LIN {X 0,Y 285.756,Z 658.565,A -85,B 0,C 180,E1 17474.349,E2 17474.349} C_VEL
LIN {X 0,Y 305.799,Z 701.656,A -85,B 0,C 180,E1 17484.152,E2 17484.152} C_VEL
LIN {X 0,Y 312.172,Z 727.073,A -85,B 0,C 180,E1 17488.423,E2 17488.423} C_VEL
LIN {X 0,Y 292.235,Z 787.027,A -85,B 0,C 180,E1 17493.812,E2 17493.812} C_VEL
LIN {X 0,Y 268.974,Z 838.866,A -85,B 0,C 180,E1 17502.314,E2 17502.314} C_VEL
LIN {X 0,Y 248.662,Z 880.297,A -85,B 0,C 180,E1 17514.564,E2 17514.564} C_VEL
LIN {X 0,Y 238.211,Z 907.781,A -85,B 0,C 180,E1 17529.488,E2 17529.488} C_VEL
LIN {X 0,Y 236.533,Z 919.61,A -85,B 0,C 180,E1 17543.125,E2 17543.125} C_VEL
LIN {X 0,Y 236.659,Z 920.093,A -85,B 0,C 180,E1 17555.518,E2 17555.518} C_VEL
LIN {X 0,Y 237.841,Z 908.97,A -85,B 0,C 180,E1 17569.569,E2 17569.569} C_VEL
LIN {X 0,Y 247.611,Z 883.003,A -85,B 0,C 180,E1 17584.7,E2 17584.7} C_VEL
LIN {X 0,Y 269.348,Z 841.838,A -85,B 0,C 180,E1 17597.744,E2 17597.744} C_VEL
LIN {X 0,Y 295.092,Z 790.298,A -85,B 0,C 180,E1 17606.682,E2 17606.682} C_VEL
LIN {X 0,Y 317.64,Z 730.915,A -85,B 0,C 180,E1 17612.277,E2 17612.277} C_VEL
LIN {X 0,Y 319.176,Z 721.636,A -85,B 0,C 180,E1 17613.218,E2 17613.218} C_VEL
LIN {X 0,Y 311.516,Z 690.262,A -85,B 0,C 180,E1 17620.895,E2 17620.895} C_VEL
LIN {X 0,Y 304.486,Z 672.096,A -85,B 0,C 180,E1 17629.77,E2 17629.77} C_VEL
LIN {X 0,Y 300.924,Z 676.866,A -85,B 0,C 180,E1 17636.437,E2 17636.437} C_VEL
LIN {X 0,Y 302.486,Z 683.644,A -85,B 0,C 180,E1 17643.411,E2 17643.411} C_VEL
LIN {X 0,Y 306.536,Z 706.136,A -85,B 0,C 180,E1 17652.005,E2 17652.005} C_VEL
LIN {X 0,Y 306.21,Z 719.511,A -85,B 0,C 180,E1 17654.903,E2 17654.903} C_VEL
LIN {X 0,Y 283.493,Z 770.529,A -85,B 0,C 180,E1 17660.967,E2 17660.967} C_VEL
LIN {X 0,Y 260.071,Z 809.733,A -85,B 0,C 180,E1 17669.993,E2 17669.993} C_VEL
LIN {X 0,Y 241.204,Z 836.353,A -85,B 0,C 180,E1 17682.29,E2 17682.29} C_VEL
LIN {X 0,Y 231.777,Z 848.177,A -85,B 0,C 180,E1 17696.186,E2 17696.186} C_VEL
LIN {X 0,Y 230.704,Z 847.604,A -85,B 0,C 180,E1 17708.792,E2 17708.792} C_VEL
LIN {X 0,Y 237.274,Z 834.196,A -85,B 0,C 180,E1 17722.816,E2 17722.816} C_VEL
LIN {X 0,Y 252.204,Z 806.032,A -85,B 0,C 180,E1 17735.424,E2 17735.424} C_VEL
LIN {X 0,Y 272.012,Z 764.995,A -85,B 0,C 180,E1 17744.744,E2 17744.744} C_VEL
LIN {X 0,Y 290.785,Z 713.245,A -85,B 0,C 180,E1 17751.027,E2 17751.027} C_VEL
LIN {X 0,Y 292.766,Z 701.675,A -85,B 0,C 180,E1 17752.282,E2 17752.282} C_VEL
LIN {X 0,Y 279.473,Z 664.949,A -85,B 0,C 180,E1 17761.189,E2 17761.189} C_VEL
LIN {X 0,Y 262.364,Z 636.414,A -85,B 0,C 180,E1 17772.063,E2 17772.063} C_VEL
LIN {X 0,Y 249.885,Z 618.017,A -85,B 0,C 180,E1 17784.7,E2 17784.7} C_VEL
LIN {X 0,Y 246.642,Z 613.282,A -85,B 0,C 180,E1 17801.641,E2 17801.641} C_VEL
LIN {X 0,Y 253.782,Z 621.283,A -85,B 0,C 180,E1 17813.984,E2 17813.984} C_VEL
LIN {X 0,Y 263.474,Z 634.294,A -85,B 0,C 180,E1 17822.404,E2 17822.404} C_VEL
LIN {X 0,Y 282.574,Z 665.228,A -85,B 0,C 180,E1 17833.721,E2 17833.721} C_VEL
LIN {X 0,Y 300.675,Z 706.247,A -85,B 0,C 180,E1 17843.349,E2 17843.349} C_VEL
LIN {X 0,Y 306.304,Z 729.368,A -85,B 0,C 180,E1 17847.452,E2 17847.452} C_VEL
LIN {X 0,Y 285.771,Z 788.355,A -85,B 0,C 180,E1 17852.891,E2 17852.891} C_VEL
LIN {X 0,Y 262.152,Z 838.88,A -85,B 0,C 180,E1 17861.401,E2 17861.401} C_VEL
LIN {X 0,Y 240.939,Z 880.256,A -85,B 0,C 180,E1 17874.076,E2 17874.076} C_VEL
LIN {X 0,Y 230.174,Z 907.605,A -85,B 0,C 180,E1 17889.748,E2 17889.748} C_VEL
LIN {X 0,Y 228.679,Z 918.896,A -85,B 0,C 180,E1 17904.286,E2 17904.286} C_VEL
LIN {X 0,Y 228.733,Z 918.872,A -85,B 0,C 180,E1 17915.71,E2 17915.71} C_VEL
LIN {X 0,Y 229.978,Z 907.706,A -85,B 0,C 180,E1 17930.267,E2 17930.267} C_VEL
LIN {X 0,Y 240.807,Z 881.536,A -85,B 0,C 180,E1 17945.935,E2 17945.935} C_VEL
LIN {X 0,Y 263.596,Z 840.67,A -85,B 0,C 180,E1 17959.097,E2 17959.097} C_VEL
LIN {X 0,Y 290.556,Z 789.057,A -85,B 0,C 180,E1 17968.069,E2 17968.069} C_VEL
LIN {X 0,Y 313.57,Z 730.598,A -85,B 0,C 180,E1 17973.545,E2 17973.545} C_VEL
LIN {X 0,Y 311.052,Z 707.647,A -85,B 0,C 180,E1 17978.228,E2 17978.228} C_VEL
LIN {X 0,Y 303.827,Z 684.399,A -85,B 0,C 180,E1 17986.891,E2 17986.891} C_VEL
LIN {X 0,Y 300.918,Z 677.004,A -85,B 0,C 180,E1 17994.813,E2 17994.813} C_VEL
LIN {X 0,Y 300.924,Z 676.866,A -85,B 0,C 180,E1 17996.437,E2 17996.437} C_VEL
LIN {X 0,Y 299.494,Z 690.532,A -85,B 0,C 180,E1 18002.762,E2 18002.762} C_VEL
LIN {X 0,Y 302.297,Z 710.977,A -85,B 0,C 180,E1 18011.066,E2 18011.066} C_VEL
LIN {X 0,Y 301.828,Z 722.39,A -85,B 0,C 180,E1 18013.737,E2 18013.737} C_VEL
LIN {X 0,Y 278.895,Z 771.501,A -85,B 0,C 180,E1 18019.625,E2 18019.625} C_VEL
LIN {X 0,Y 254.375,Z 810.659,A -85,B 0,C 180,E1 18028.68,E2 18028.68} C_VEL
LIN {X 0,Y 234.95,Z 836.493,A -85,B 0,C 180,E1 18040.585,E2 18040.585} C_VEL
LIN {X 0,Y 224.337,Z 849.161,A -85,B 0,C 180,E1 18054.904,E2 18054.904} C_VEL
LIN {X 0,Y 223.072,Z 848.185,A -85,B 0,C 180,E1 18070.116,E2 18070.116} C_VEL
LIN {X 0,Y 230.402,Z 834.015,A -85,B 0,C 180,E1 18084.332,E2 18084.332} C_VEL
LIN {X 0,Y 246.032,Z 806.043,A -85,B 0,C 180,E1 18096.737,E2 18096.737} C_VEL
LIN {X 0,Y 266.699,Z 764.716,A -85,B 0,C 180,E1 18106.106,E2 18106.106} C_VEL
LIN {X 0,Y 286.019,Z 712.916,A -85,B 0,C 180,E1 18112.334,E2 18112.334} C_VEL
LIN {X 0,Y 286.388,Z 701.757,A -85,B 0,C 180,E1 18114.013,E2 18114.013} C_VEL
LIN {X 0,Y 273.45,Z 666.448,A -85,B 0,C 180,E1 18123.313,E2 18123.313} C_VEL
LIN {X 0,Y 257.524,Z 639.288,A -85,B 0,C 180,E1 18134.83,E2 18134.83} C_VEL
LIN {X 0,Y 247.315,Z 625.136,A -85,B 0,C 180,E1 18147.059,E2 18147.059} C_VEL
LIN {X 0,Y 245.601,Z 621.305,A -85,B 0,C 180,E1 18161.71,E2 18161.71} C_VEL
LIN {X 0,Y 252.429,Z 629.123,A -85,B 0,C 180,E1 18173.688,E2 18173.688} C_VEL
LIN {X 0,Y 263.127,Z 644.042,A -85,B 0,C 180,E1 18183.035,E2 18183.035} C_VEL
LIN {X 0,Y 281.121,Z 675.674,A -85,B 0,C 180,E1 18194.191,E2 18194.191} C_VEL
LIN {X 0,Y 297.749,Z 717.835,A -85,B 0,C 180,E1 18203.991,E2 18203.991} C_VEL
LIN {X 0,Y 300.028,Z 733.449,A -85,B 0,C 180,E1 18206.564,E2 18206.564} C_VEL
LIN {X 0,Y 277.496,Z 793.955,A -85,B 0,C 180,E1 18212.487,E2 18212.487} C_VEL
LIN {X 0,Y 252.286,Z 844.934,A -85,B 0,C 180,E1 18221.893,E2 18221.893} C_VEL
LIN {X 0,Y 231.41,Z 884.207,A -85,B 0,C 180,E1 18235.349,E2 18235.349} C_VEL
LIN {X 0,Y 221.734,Z 909.528,A -85,B 0,C 180,E1 18252.061,E2 18252.061} C_VEL
LIN {X 0,Y 220.778,Z 917.691,A -85,B 0,C 180,E1 18264.239,E2 18264.239} C_VEL
LIN {X 0,Y 220.79,Z 917.646,A -85,B 0,C 180,E1 18275.916,E2 18275.916} C_VEL
LIN {X 0,Y 222.201,Z 906.459,A -85,B 0,C 180,E1 18291.009,E2 18291.009} C_VEL
LIN {X 0,Y 233.986,Z 880.303,A -85,B 0,C 180,E1 18307.148,E2 18307.148} C_VEL
LIN {X 0,Y 258.018,Z 839.639,A -85,B 0,C 180,E1 18320.481,E2 18320.481} C_VEL
LIN {X 0,Y 285.967,Z 788.348,A -85,B 0,C 180,E1 18329.436,E2 18329.436} C_VEL
LIN {X 0,Y 309.296,Z 729.164,A -85,B 0,C 180,E1 18335.183,E2 18335.183} C_VEL
LIN {X 0,Y 304.166,Z 701.793,A -85,B 0,C 180,E1 18342.646,E2 18342.646} C_VEL
LIN {X 0,Y 299.965,Z 687.774,A -85,B 0,C 180,E1 18349.861,E2 18349.861} C_VEL
LIN {X 0,Y 298.698,Z 685.744,A -85,B 0,C 180,E1 18358.601,E2 18358.601} C_VEL
LIN {X 0,Y 299.494,Z 690.532,A -85,B 0,C 180,E1 18362.762,E2 18362.762} C_VEL
LIN {X 0,Y 297.796,Z 710.81,A -85,B 0,C 180,E1 18368.411,E2 18368.411} C_VEL
LIN {X 0,Y 296.984,Z 726.69,A -85,B 0,C 180,E1 18372.665,E2 18372.665} C_VEL
LIN {X 0,Y 272.134,Z 776.524,A -85,B 0,C 180,E1 18378.912,E2 18378.912} C_VEL
LIN {X 0,Y 246.056,Z 815.395,A -85,B 0,C 180,E1 18388.594,E2 18388.594} C_VEL
LIN {X 0,Y 225.73,Z 840.486,A -85,B 0,C 180,E1 18401.706,E2 18401.706} C_VEL
LIN {X 0,Y 216.947,Z 850.083,A -85,B 0,C 180,E1 18413.651,E2 18413.651} C_VEL
LIN {X 0,Y 214.574,Z 850.715,A -85,B 0,C 180,E1 18427.111,E2 18427.111} C_VEL
LIN {X 0,Y 220.669,Z 839.38,A -85,B 0,C 180,E1 18441.914,E2 18441.914} C_VEL
LIN {X 0,Y 235.858,Z 813.54,A -85,B 0,C 180,E1 18455.54,E2 18455.54} C_VEL
LIN {X 0,Y 256.152,Z 775.907,A -85,B 0,C 180,E1 18465.463,E2 18465.463} C_VEL
LIN {X 0,Y 276.694,Z 726.885,A -85,B 0,C 180,E1 18472.365,E2 18472.365} C_VEL
LIN {X 0,Y 281.668,Z 708.955,A -85,B 0,C 180,E1 18474.219,E2 18474.219} C_VEL
LIN {X 0,Y 270.443,Z 674.474,A -85,B 0,C 180,E1 18483.46,E2 18483.46} C_VEL
LIN {X 0,Y 255.662,Z 646.909,A -85,B 0,C 180,E1 18495.168,E2 18495.168} C_VEL
LIN {X 0,Y 246.004,Z 632.903,A -85,B 0,C 180,E1 18507.493,E2 18507.493} C_VEL
LIN {X 0,Y 244.573,Z 629.3,A -85,B 0,C 180,E1 18521.809,E2 18521.809} C_VEL
LIN {X 0,Y 251.076,Z 636.937,A -85,B 0,C 180,E1 18533.379,E2 18533.379} C_VEL
LIN {X 0,Y 262.218,Z 653.044,A -85,B 0,C 180,E1 18543.357,E2 18543.357} C_VEL
LIN {X 0,Y 279.482,Z 686.4,A -85,B 0,C 180,E1 18554.778,E2 18554.778} C_VEL
LIN {X 0,Y 293.957,Z 728.626,A -85,B 0,C 180,E1 18564.483,E2 18564.483} C_VEL
LIN {X 0,Y 293.002,Z 739.507,A -85,B 0,C 180,E1 18565.829,E2 18565.829} C_VEL
LIN {X 0,Y 270.413,Z 796.506,A -85,B 0,C 180,E1 18571.696,E2 18571.696} C_VEL
LIN {X 0,Y 244.727,Z 846.193,A -85,B 0,C 180,E1 18581.271,E2 18581.271} C_VEL
LIN {X 0,Y 223.718,Z 883.939,A -85,B 0,C 180,E1 18594.788,E2 18594.788} C_VEL
LIN {X 0,Y 213.898,Z 908.137,A -85,B 0,C 180,E1 18611.38,E2 18611.38} C_VEL
LIN {X 0,Y 212.809,Z 916.386,A -85,B 0,C 180,E1 18623.858,E2 18623.858} C_VEL
LIN {X 0,Y 212.842,Z 916.424,A -85,B 0,C 180,E1 18636.137,E2 18636.137} C_VEL
LIN {X 0,Y 214.121,Z 906.378,A -85,B 0,C 180,E1 18650.752,E2 18650.752} C_VEL
LIN {X 0,Y 226.469,Z 880.45,A -85,B 0,C 180,E1 18667.808,E2 18667.808} C_VEL
LIN {X 0,Y 251.768,Z 839.926,A -85,B 0,C 180,E1 18681.619,E2 18681.619} C_VEL
LIN {X 0,Y 281.142,Z 788.507,A -85,B 0,C 180,E1 18690.754,E2 18690.754} C_VEL
LIN {X 0,Y 304.387,Z 732.594,A -85,B 0,C 180,E1 18696.267,E2 18696.267} C_VEL
LIN {X 0,Y 300.184,Z 706.471,A -85,B 0,C 180,E1 18703.921,E2 18703.921} C_VEL
LIN {X 0,Y 296.811,Z 694.336,A -85,B 0,C 180,E1 18711.2,E2 18711.2} C_VEL
LIN {X 0,Y 296.088,Z 693.324,A -85,B 0,C 180,E1 18718.588,E2 18718.588} C_VEL
LIN {X 0,Y 297.437,Z 706.176,A -85,B 0,C 180,E1 18726.645,E2 18726.645} C_VEL
LIN {X 0,Y 297.796,Z 710.81,A -85,B 0,C 180,E1 18728.411,E2 18728.411} C_VEL
LIN {X 0,Y 295.364,Z 723.191,A -85,B 0,C 180,E1 18730.755,E2 18730.755} C_VEL
LIN {X 0,Y 288.736,Z 738.824,A -85,B 0,C 180,E1 18732.316,E2 18732.316} C_VEL
LIN {X 0,Y 262.641,Z 785.694,A -85,B 0,C 180,E1 18738.979,E2 18738.979} C_VEL
LIN {X 0,Y 236.659,Z 821.229,A -85,B 0,C 180,E1 18749.008,E2 18749.008} C_VEL
LIN {X 0,Y 216.724,Z 843.948,A -85,B 0,C 180,E1 18762.677,E2 18762.677} C_VEL
LIN {X 0,Y 207.622,Z 852.599,A -85,B 0,C 180,E1 18777.309,E2 18777.309} C_VEL
LIN {X 0,Y 208.233,Z 848.927,A -85,B 0,C 180,E1 18793.399,E2 18793.399} C_VEL
LIN {X 0,Y 218.395,Z 831.675,A -85,B 0,C 180,E1 18808.674,E2 18808.674} C_VEL
LIN {X 0,Y 237.945,Z 799.409,A -85,B 0,C 180,E1 18821.498,E2 18821.498} C_VEL
LIN {X 0,Y 261.063,Z 754.132,A -85,B 0,C 180,E1 18830.5,E2 18830.5} C_VEL
LIN {X 0,Y 276,Z 711.618,A -85,B 0,C 180,E1 18835.458,E2 18835.458} C_VEL
LIN {X 0,Y 265.972,Z 679.01,A -85,B 0,C 180,E1 18844.683,E2 18844.683} C_VEL
LIN {X 0,Y 252.607,Z 653.366,A -85,B 0,C 180,E1 18856.406,E2 18856.406} C_VEL
LIN {X 0,Y 244.487,Z 640.557,A -85,B 0,C 180,E1 18868.092,E2 18868.092} C_VEL
LIN {X 0,Y 243.496,Z 637.271,A -85,B 0,C 180,E1 18881.78,E2 18881.78} C_VEL
LIN {X 0,Y 249.831,Z 645.112,A -85,B 0,C 180,E1 18893.374,E2 18893.374} C_VEL
LIN {X 0,Y 260.201,Z 661.255,A -85,B 0,C 180,E1 18903.174,E2 18903.174} C_VEL
LIN {X 0,Y 275.808,Z 693.161,A -85,B 0,C 180,E1 18914.267,E2 18914.267} C_VEL
LIN {X 0,Y 289.1,Z 735.715,A -85,B 0,C 180,E1 18924.293,E2 18924.293} C_VEL
LIN {X 0,Y 265.502,Z 794.732,A -85,B 0,C 180,E1 18930.261,E2 18930.261} C_VEL
LIN {X 0,Y 238.86,Z 844.483,A -85,B 0,C 180,E1 18939.809,E2 18939.809} C_VEL
LIN {X 0,Y 216.77,Z 882.281,A -85,B 0,C 180,E1 18953.481,E2 18953.481} C_VEL
LIN {X 0,Y 206.069,Z 906.722,A -85,B 0,C 180,E1 18970.645,E2 18970.645} C_VEL
LIN {X 0,Y 204.869,Z 915.125,A -85,B 0,C 180,E1 18983.619,E2 18983.619} C_VEL
LIN {X 0,Y 204.89,Z 915.198,A -85,B 0,C 180,E1 18996.377,E2 18996.377} C_VEL
LIN {X 0,Y 206.365,Z 905.146,A -85,B 0,C 180,E1 19011.57,E2 19011.57} C_VEL
LIN {X 0,Y 219.047,Z 880.402,A -85,B 0,C 180,E1 19028.57,E2 19028.57} C_VEL
LIN {X 0,Y 245.447,Z 840.432,A -85,B 0,C 180,E1 19042.749,E2 19042.749} C_VEL
LIN {X 0,Y 275.715,Z 790.077,A -85,B 0,C 180,E1 19051.919,E2 19051.919} C_VEL
LIN {X 0,Y 299.55,Z 735.967,A -85,B 0,C 180,E1 19057.414,E2 19057.414} C_VEL
LIN {X 0,Y 296.354,Z 711.703,A -85,B 0,C 180,E1 19065.079,E2 19065.079} C_VEL
LIN {X 0,Y 293.659,Z 700.98,A -85,B 0,C 180,E1 19072.637,E2 19072.637} C_VEL
LIN {X 0,Y 293.308,Z 701.695,A -85,B 0,C 180,E1 19079.686,E2 19079.686} C_VEL
LIN {X 0,Y 293.87,Z 718.198,A -85,B 0,C 180,E1 19088.218,E2 19088.218} C_VEL
LIN {X 0,Y 292.904,Z 729.47,A -85,B 0,C 180,E1 19091.416,E2 19091.416} C_VEL
LIN {X 0,Y 288.736,Z 738.824,A -85,B 0,C 180,E1 19092.316,E2 19092.316} C_VEL
LIN {X 0,Y 270.495,Z 767.731,A -85,B 0,C 180,E1 19094.242,E2 19094.242} C_VEL
LIN {X 0,Y 241.389,Z 809.699,A -85,B 0,C 180,E1 19103.087,E2 19103.087} C_VEL
LIN {X 0,Y 216.003,Z 838.571,A -85,B 0,C 180,E1 19116.109,E2 19116.109} C_VEL
LIN {X 0,Y 201.698,Z 852.529,A -85,B 0,C 180,E1 19132.289,E2 19132.289} C_VEL
LIN {X 0,Y 199.239,Z 852.145,A -85,B 0,C 180,E1 19149.958,E2 19149.958} C_VEL
LIN {X 0,Y 207.662,Z 838.172,A -85,B 0,C 180,E1 19165.996,E2 19165.996} C_VEL
LIN {X 0,Y 225.755,Z 810.237,A -85,B 0,C 180,E1 19179.676,E2 19179.676} C_VEL
LIN {X 0,Y 249.087,Z 769.143,A -85,B 0,C 180,E1 19189.579,E2 19189.579} C_VEL
LIN {X 0,Y 270.747,Z 716.234,A -85,B 0,C 180,E1 19196.272,E2 19196.272} C_VEL
LIN {X 0,Y 261.838,Z 684.683,A -85,B 0,C 180,E1 19205.577,E2 19205.577} C_VEL
LIN {X 0,Y 249.851,Z 660.2,A -85,B 0,C 180,E1 19217.308,E2 19217.308} C_VEL
LIN {X 0,Y 243.013,Z 648.329,A -85,B 0,C 180,E1 19228.416,E2 19228.416} C_VEL
LIN {X 0,Y 242.244,Z 645.163,A -85,B 0,C 180,E1 19241.682,E2 19241.682} C_VEL
LIN {X 0,Y 248.26,Z 652.931,A -85,B 0,C 180,E1 19253.134,E2 19253.134} C_VEL
LIN {X 0,Y 258.601,Z 670.439,A -85,B 0,C 180,E1 19263.509,E2 19263.509} C_VEL
LIN {X 0,Y 273.157,Z 703.222,A -85,B 0,C 180,E1 19274.717,E2 19274.717} C_VEL
LIN {X 0,Y 283.014,Z 739.353,A -85,B 0,C 180,E1 19283.325,E2 19283.325} C_VEL
LIN {X 0,Y 258.862,Z 796.578,A -85,B 0,C 180,E1 19289.293,E2 19289.293} C_VEL
LIN {X 0,Y 231.377,Z 845.745,A -85,B 0,C 180,E1 19299.111,E2 19299.111} C_VEL
LIN {X 0,Y 208.218,Z 883.681,A -85,B 0,C 180,E1 19313.765,E2 19313.765} C_VEL
LIN {X 0,Y 197.836,Z 907.082,A -85,B 0,C 180,E1 19331.838,E2 19331.838} C_VEL
LIN {X 0,Y 196.92,Z 913.86,A -85,B 0,C 180,E1 19343.36,E2 19343.36} C_VEL
LIN {X 0,Y 196.939,Z 913.978,A -85,B 0,C 180,E1 19356.635,E2 19356.635} C_VEL
LIN {X 0,Y 198.618,Z 903.937,A -85,B 0,C 180,E1 19372.439,E2 19372.439} C_VEL
LIN {X 0,Y 213.893,Z 877.227,A -85,B 0,C 180,E1 19391.013,E2 19391.013} C_VEL
LIN {X 0,Y 242.601,Z 836.075,A -85,B 0,C 180,E1 19405.182,E2 19405.182} C_VEL
LIN {X 0,Y 273.786,Z 785.568,A -85,B 0,C 180,E1 19413.936,E2 19413.936} C_VEL
LIN {X 0,Y 294.864,Z 739.603,A -85,B 0,C 180,E1 19418.541,E2 19418.541} C_VEL
LIN {X 0,Y 292.615,Z 717.385,A -85,B 0,C 180,E1 19426.008,E2 19426.008} C_VEL
LIN {X 0,Y 290.74,Z 708.502,A -85,B 0,C 180,E1 19432.563,E2 19432.563} C_VEL
LIN {X 0,Y 290.169,Z 709.729,A -85,B 0,C 180,E1 19440.057,E2 19440.057} C_VEL
LIN {X 0,Y 289.718,Z 726.409,A -85,B 0,C 180,E1 19448.336,E2 19448.336} C_VEL
LIN {X 0,Y 287.825,Z 735.017,A -85,B 0,C 180,E1 19450.378,E2 19450.378} C_VEL
LIN {X 0,Y 270.495,Z 767.731,A -85,B 0,C 180,E1 19454.242,E2 19454.242} C_VEL
LIN {X 0,Y 250.107,Z 793.576,A -85,B 0,C 180,E1 19457.134,E2 19457.134} C_VEL
LIN {X 0,Y 221.972,Z 827.261,A -85,B 0,C 180,E1 19467.736,E2 19467.736} C_VEL
LIN {X 0,Y 200.987,Z 848.055,A -85,B 0,C 180,E1 19482.247,E2 19482.247} C_VEL
LIN {X 0,Y 191.333,Z 855.421,A -85,B 0,C 180,E1 19498.969,E2 19498.969} C_VEL
LIN {X 0,Y 193.424,Z 850.005,A -85,B 0,C 180,E1 19516.102,E2 19516.102} C_VEL
LIN {X 0,Y 205.976,Z 831.105,A -85,B 0,C 180,E1 19532.113,E2 19532.113} C_VEL
LIN {X 0,Y 228.041,Z 797.623,A -85,B 0,C 180,E1 19545.028,E2 19545.028} C_VEL
LIN {X 0,Y 252.379,Z 752.096,A -85,B 0,C 180,E1 19553.712,E2 19553.712} C_VEL
LIN {X 0,Y 265.147,Z 718.704,A -85,B 0,C 180,E1 19557.661,E2 19557.661} C_VEL
LIN {X 0,Y 257.149,Z 688.712,A -85,B 0,C 180,E1 19567.109,E2 19567.109} C_VEL
LIN {X 0,Y 246.257,Z 665.176,A -85,B 0,C 180,E1 19579.353,E2 19579.353} C_VEL
LIN {X 0,Y 240.962,Z 655.607,A -85,B 0,C 180,E1 19589.679,E2 19589.679} C_VEL
LIN {X 0,Y 241.059,Z 653.334,A -85,B 0,C 180,E1 19602.52,E2 19602.52} C_VEL
LIN {X 0,Y 246.878,Z 661.288,A -85,B 0,C 180,E1 19613.428,E2 19613.428} C_VEL
LIN {X 0,Y 257.285,Z 680.476,A -85,B 0,C 180,E1 19624.302,E2 19624.302} C_VEL
LIN {X 0,Y 270.372,Z 713.971,A -85,B 0,C 180,E1 19635.392,E2 19635.392} C_VEL
LIN {X 0,Y 276.748,Z 743.456,A -85,B 0,C 180,E1 19642.336,E2 19642.336} C_VEL
LIN {X 0,Y 250.186,Z 802.451,A -85,B 0,C 180,E1 19648.867,E2 19648.867} C_VEL
LIN {X 0,Y 221.117,Z 851.37,A -85,B 0,C 180,E1 19659.668,E2 19659.668} C_VEL
LIN {X 0,Y 198.765,Z 886.716,A -85,B 0,C 180,E1 19675.065,E2 19675.065} C_VEL
LIN {X 0,Y 189.538,Z 907.714,A -85,B 0,C 180,E1 19693.724,E2 19693.724} C_VEL
LIN {X 0,Y 189.189,Z 913.609,A -85,B 0,C 180,E1 19707.699,E2 19707.699} C_VEL
LIN {X 0,Y 189.073,Z 910.974,A -85,B 0,C 180,E1 19721.573,E2 19721.573} C_VEL
LIN {X 0,Y 195.765,Z 893.842,A -85,B 0,C 180,E1 19741.482,E2 19741.482} C_VEL
LIN {X 0,Y 219.341,Z 860.389,A -85,B 0,C 180,E1 19759.236,E2 19759.236} C_VEL
LIN {X 0,Y 251.526,Z 815.126,A -85,B 0,C 180,E1 19771.02,E2 19771.02} C_VEL
LIN {X 0,Y 282.687,Z 760.579,A -85,B 0,C 180,E1 19778.091,E2 19778.091} C_VEL
LIN {X 0,Y 290.144,Z 743.17,A -85,B 0,C 180,E1 19779.714,E2 19779.714} C_VEL
LIN {X 0,Y 288.712,Z 722.354,A -85,B 0,C 180,E1 19787.396,E2 19787.396} C_VEL
LIN {X 0,Y 287.328,Z 714.491,A -85,B 0,C 180,E1 19795.516,E2 19795.516} C_VEL
LIN {X 0,Y 286.365,Z 721.812,A -85,B 0,C 180,E1 19803.094,E2 19803.094} C_VEL
LIN {X 0,Y 284.254,Z 737.403,A -85,B 0,C 180,E1 19809.027,E2 19809.027} C_VEL
LIN {X 0,Y 255.641,Z 785.887,A -85,B 0,C 180,E1 19815.554,E2 19815.554} C_VEL
LIN {X 0,Y 250.107,Z 793.576,A -85,B 0,C 180,E1 19817.134,E2 19817.134} C_VEL
LIN {X 0,Y 228.332,Z 815.849,A -85,B 0,C 180,E1 19821.189,E2 19821.189} C_VEL
LIN {X 0,Y 201.736,Z 842.385,A -85,B 0,C 180,E1 19834.429,E2 19834.429} C_VEL
LIN {X 0,Y 185.809,Z 855.549,A -85,B 0,C 180,E1 19852.23,E2 19852.23} C_VEL
LIN {X 0,Y 183.034,Z 855.345,A -85,B 0,C 180,E1 19868.096,E2 19868.096} C_VEL
LIN {X 0,Y 191.796,Z 842.171,A -85,B 0,C 180,E1 19886.31,E2 19886.31} C_VEL
LIN {X 0,Y 211.547,Z 814.424,A -85,B 0,C 180,E1 19901.379,E2 19901.379} C_VEL
LIN {X 0,Y 237.208,Z 773.285,A -85,B 0,C 180,E1 19911.943,E2 19911.943} C_VEL
LIN {X 0,Y 259.669,Z 721.968,A -85,B 0,C 180,E1 19918.899,E2 19918.899} C_VEL
LIN {X 0,Y 252.565,Z 693.367,A -85,B 0,C 180,E1 19928.472,E2 19928.472} C_VEL
LIN {X 0,Y 242.854,Z 670.193,A -85,B 0,C 180,E1 19941.437,E2 19941.437} C_VEL
LIN {X 0,Y 238.637,Z 662.259,A -85,B 0,C 180,E1 19952.278,E2 19952.278} C_VEL
LIN {X 0,Y 239.809,Z 661.782,A -85,B 0,C 180,E1 19963.712,E2 19963.712} C_VEL
LIN {X 0,Y 246.12,Z 670.412,A -85,B 0,C 180,E1 19974.739,E2 19974.739} C_VEL
LIN {X 0,Y 257.459,Z 695.254,A -85,B 0,C 180,E1 19986.911,E2 19986.911} C_VEL
LIN {X 0,Y 268.989,Z 732.061,A -85,B 0,C 180,E1 19998.004,E2 19998.004} C_VEL
LIN {X 0,Y 270.48,Z 747.379,A -85,B 0,C 180,E1 20001.313,E2 20001.313} C_VEL
LIN {X 0,Y 243.373,Z 804.437,A -85,B 0,C 180,E1 20007.875,E2 20007.875} C_VEL
LIN {X 0,Y 214.41,Z 851.203,A -85,B 0,C 180,E1 20018.524,E2 20018.524} C_VEL
LIN {X 0,Y 190.882,Z 886.637,A -85,B 0,C 180,E1 20034.657,E2 20034.657} C_VEL
LIN {X 0,Y 181.623,Z 906.698,A -85,B 0,C 180,E1 20053.514,E2 20053.514} C_VEL
LIN {X 0,Y 181.251,Z 912.366,A -85,B 0,C 180,E1 20067.599,E2 20067.599} C_VEL
LIN {X 0,Y 181.153,Z 909.757,A -85,B 0,C 180,E1 20082.086,E2 20082.086} C_VEL
LIN {X 0,Y 188.23,Z 893.2,A -85,B 0,C 180,E1 20102.367,E2 20102.367} C_VEL
LIN {X 0,Y 212.986,Z 860.402,A -85,B 0,C 180,E1 20120.565,E2 20120.565} C_VEL
LIN {X 0,Y 246.811,Z 815.338,A -85,B 0,C 180,E1 20132.516,E2 20132.516} C_VEL
LIN {X 0,Y 279.036,Z 761.275,A -85,B 0,C 180,E1 20139.536,E2 20139.536} C_VEL
LIN {X 0,Y 285.535,Z 746.355,A -85,B 0,C 180,E1 20141.056,E2 20141.056} C_VEL
LIN {X 0,Y 284.881,Z 728.3,A -85,B 0,C 180,E1 20148.273,E2 20148.273} C_VEL
LIN {X 0,Y 284.015,Z 721.819,A -85,B 0,C 180,E1 20155.463,E2 20155.463} C_VEL
LIN {X 0,Y 282.505,Z 729.376,A -85,B 0,C 180,E1 20163.137,E2 20163.137} C_VEL
LIN {X 0,Y 279.685,Z 742.081,A -85,B 0,C 180,E1 20167.853,E2 20167.853} C_VEL
LIN {X 0,Y 250.333,Z 789.09,A -85,B 0,C 180,E1 20174.353,E2 20174.353} C_VEL
LIN {X 0,Y 228.332,Z 815.849,A -85,B 0,C 180,E1 20181.189,E2 20181.189} C_VEL
LIN {X 0,Y 206.378,Z 834.089,A -85,B 0,C 180,E1 20186.775,E2 20186.775} C_VEL
LIN {X 0,Y 184.461,Z 852.565,A -85,B 0,C 180,E1 20202.578,E2 20202.578} C_VEL
LIN {X 0,Y 175.056,Z 857.871,A -85,B 0,C 180,E1 20221.527,E2 20221.527} C_VEL
LIN {X 0,Y 179.705,Z 849.779,A -85,B 0,C 180,E1 20240.534,E2 20240.534} C_VEL
LIN {X 0,Y 196.477,Z 827.567,A -85,B 0,C 180,E1 20257.38,E2 20257.38} C_VEL
LIN {X 0,Y 220.878,Z 792.638,A -85,B 0,C 180,E1 20269.57,E2 20269.57} C_VEL
LIN {X 0,Y 247.057,Z 744.391,A -85,B 0,C 180,E1 20277.825,E2 20277.825} C_VEL
LIN {X 0,Y 254.36,Z 725.799,A -85,B 0,C 180,E1 20280.018,E2 20280.018} C_VEL
LIN {X 0,Y 248.014,Z 697.668,A -85,B 0,C 180,E1 20290.031,E2 20290.031} C_VEL
LIN {X 0,Y 239.756,Z 676.832,A -85,B 0,C 180,E1 20302.757,E2 20302.757} C_VEL
LIN {X 0,Y 236.582,Z 669.345,A -85,B 0,C 180,E1 20313.888,E2 20313.888} C_VEL
LIN {X 0,Y 238.204,Z 670.102,A -85,B 0,C 180,E1 20324.698,E2 20324.698} C_VEL
LIN {X 0,Y 244.284,Z 678.932,A -85,B 0,C 180,E1 20335.145,E2 20335.145} C_VEL
LIN {X 0,Y 255.016,Z 705.471,A -85,B 0,C 180,E1 20347.621,E2 20347.621} C_VEL
LIN {X 0,Y 264.614,Z 741.037,A -85,B 0,C 180,E1 20358.312,E2 20358.312} C_VEL
LIN {X 0,Y 264.265,Z 751.182,A -85,B 0,C 180,E1 20360.271,E2 20360.271} C_VEL
LIN {X 0,Y 236.709,Z 806.27,A -85,B 0,C 180,E1 20366.798,E2 20366.798} C_VEL
LIN {X 0,Y 206.607,Z 852.684,A -85,B 0,C 180,E1 20377.85,E2 20377.85} C_VEL
LIN {X 0,Y 182.784,Z 886.916,A -85,B 0,C 180,E1 20394.465,E2 20394.465} C_VEL
LIN {X 0,Y 173.44,Z 906.824,A -85,B 0,C 180,E1 20415.288,E2 20415.288} C_VEL
LIN {X 0,Y 173.321,Z 911.123,A -85,B 0,C 180,E1 20427.489,E2 20427.489} C_VEL
LIN {X 0,Y 173.216,Z 908.538,A -85,B 0,C 180,E1 20442.649,E2 20442.649} C_VEL
LIN {X 0,Y 181.104,Z 891.995,A -85,B 0,C 180,E1 20463.807,E2 20463.807} C_VEL
LIN {X 0,Y 207.775,Z 859.089,A -85,B 0,C 180,E1 20482.495,E2 20482.495} C_VEL
LIN {X 0,Y 243.861,Z 813.316,A -85,B 0,C 180,E1 20494.461,E2 20494.461} C_VEL
LIN {X 0,Y 277.127,Z 758.894,A -85,B 0,C 180,E1 20501.3,E2 20501.3} C_VEL
LIN {X 0,Y 281.078,Z 748.604,A -85,B 0,C 180,E1 20502.795,E2 20502.795} C_VEL
LIN {X 0,Y 280.83,Z 732.432,A -85,B 0,C 180,E1 20510.57,E2 20510.57} C_VEL
LIN {X 0,Y 280.438,Z 729.013,A -85,B 0,C 180,E1 20515.405,E2 20515.405} C_VEL
LIN {X 0,Y 278.314,Z 736.889,A -85,B 0,C 180,E1 20523.184,E2 20523.184} C_VEL
LIN {X 0,Y 275.63,Z 746.202,A -85,B 0,C 180,E1 20526.587,E2 20526.587} C_VEL
LIN {X 0,Y 243.618,Z 794.199,A -85,B 0,C 180,E1 20533.484,E2 20533.484} C_VEL
LIN {X 0,Y 212.338,Z 828.552,A -85,B 0,C 180,E1 20544.062,E2 20544.062} C_VEL
LIN {X 0,Y 206.378,Z 834.089,A -85,B 0,C 180,E1 20546.775,E2 20546.775} C_VEL
LIN {X 0,Y 185.449,Z 847.926,A -85,B 0,C 180,E1 20554.116,E2 20554.116} C_VEL
LIN {X 0,Y 171.663,Z 857.509,A -85,B 0,C 180,E1 20568.833,E2 20568.833} C_VEL
LIN {X 0,Y 167.024,Z 858.455,A -85,B 0,C 180,E1 20585.87,E2 20585.87} C_VEL
LIN {X 0,Y 175.205,Z 846.819,A -85,B 0,C 180,E1 20605.802,E2 20605.802} C_VEL
LIN {X 0,Y 195.778,Z 820.95,A -85,B 0,C 180,E1 20622.31,E2 20622.31} C_VEL
LIN {X 0,Y 222.774,Z 782.095,A -85,B 0,C 180,E1 20633.606,E2 20633.606} C_VEL
LIN {X 0,Y 248.568,Z 731.886,A -85,B 0,C 180,E1 20640.793,E2 20640.793} C_VEL
LIN {X 0,Y 245.533,Z 709.104,A -85,B 0,C 180,E1 20648.46,E2 20648.46} C_VEL
LIN {X 0,Y 238.101,Z 686.696,A -85,B 0,C 180,E1 20660.934,E2 20660.934} C_VEL
LIN {X 0,Y 234.603,Z 677.958,A -85,B 0,C 180,E1 20671.759,E2 20671.759} C_VEL
LIN {X 0,Y 235.72,Z 677.102,A -85,B 0,C 180,E1 20683.293,E2 20683.293} C_VEL
LIN {X 0,Y 241.56,Z 686.133,A -85,B 0,C 180,E1 20694.634,E2 20694.634} C_VEL
LIN {X 0,Y 251.111,Z 712.075,A -85,B 0,C 180,E1 20707.087,E2 20707.087} C_VEL
LIN {X 0,Y 259.381,Z 746.786,A -85,B 0,C 180,E1 20717.813,E2 20717.813} C_VEL
LIN {X 0,Y 257.329,Z 756.657,A -85,B 0,C 180,E1 20719.319,E2 20719.319} C_VEL
LIN {X 0,Y 227.507,Z 812.372,A -85,B 0,C 180,E1 20726.445,E2 20726.445} C_VEL
LIN {X 0,Y 197.053,Z 856.578,A -85,B 0,C 180,E1 20738.044,E2 20738.044} C_VEL
LIN {X 0,Y 173.026,Z 889.649,A -85,B 0,C 180,E1 20756.221,E2 20756.221} C_VEL
LIN {X 0,Y 165.387,Z 906.576,A -85,B 0,C 180,E1 20776.736,E2 20776.736} C_VEL
LIN {X 0,Y 165.44,Z 909.995,A -85,B 0,C 180,E1 20792.626,E2 20792.626} C_VEL
LIN {X 0,Y 165.823,Z 904.641,A -85,B 0,C 180,E1 20808.679,E2 20808.679} C_VEL
LIN {X 0,Y 178.965,Z 884.504,A -85,B 0,C 180,E1 20830.467,E2 20830.467} C_VEL
LIN {X 0,Y 209.826,Z 850.016,A -85,B 0,C 180,E1 20847.26,E2 20847.26} C_VEL
LIN {X 0,Y 247.714,Z 802.351,A -85,B 0,C 180,E1 20857.902,E2 20857.902} C_VEL
LIN {X 0,Y 276.386,Z 754.607,A -85,B 0,C 180,E1 20863.33,E2 20863.33} C_VEL
LIN {X 0,Y 276.923,Z 739.573,A -85,B 0,C 180,E1 20870.602,E2 20870.602} C_VEL
LIN {X 0,Y 276.667,Z 736.129,A -85,B 0,C 180,E1 20875.343,E2 20875.343} C_VEL
LIN {X 0,Y 274.267,Z 742.86,A -85,B 0,C 180,E1 20882.438,E2 20882.438} C_VEL
LIN {X 0,Y 271.649,Z 750.321,A -85,B 0,C 180,E1 20885.296,E2 20885.296} C_VEL
LIN {X 0,Y 240.238,Z 795.258,A -85,B 0,C 180,E1 20891.744,E2 20891.744} C_VEL
LIN {X 0,Y 207.142,Z 829.916,A -85,B 0,C 180,E1 20902.399,E2 20902.399} C_VEL
LIN {X 0,Y 185.449,Z 847.926,A -85,B 0,C 180,E1 20914.116,E2 20914.116} C_VEL
LIN {X 0,Y 167.272,Z 857.076,A -85,B 0,C 180,E1 20923.607,E2 20923.607} C_VEL
LIN {X 0,Y 159.09,Z 859.789,A -85,B 0,C 180,E1 20945.181,E2 20945.181} C_VEL
LIN {X 0,Y 166.951,Z 849.044,A -85,B 0,C 180,E1 20965.594,E2 20965.594} C_VEL
LIN {X 0,Y 187.932,Z 823.988,A -85,B 0,C 180,E1 20982.848,E2 20982.848} C_VEL
LIN {X 0,Y 215.496,Z 786.462,A -85,B 0,C 180,E1 20994.493,E2 20994.493} C_VEL
LIN {X 0,Y 242.371,Z 737.216,A -85,B 0,C 180,E1 21001.907,E2 21001.907} C_VEL
LIN {X 0,Y 243.381,Z 727.475,A -85,B 0,C 180,E1 21004.365,E2 21004.365} C_VEL
LIN {X 0,Y 238.202,Z 703.517,A -85,B 0,C 180,E1 21014.925,E2 21014.925} C_VEL
LIN {X 0,Y 233.438,Z 688.606,A -85,B 0,C 180,E1 21026.387,E2 21026.387} C_VEL
LIN {X 0,Y 233.031,Z 684.048,A -85,B 0,C 180,E1 21041.471,E2 21041.471} C_VEL
LIN {X 0,Y 238.34,Z 692.735,A -85,B 0,C 180,E1 21053.718,E2 21053.718} C_VEL
LIN {X 0,Y 247.087,Z 718.569,A -85,B 0,C 180,E1 21066.542,E2 21066.542} C_VEL
LIN {X 0,Y 254.014,Z 752.235,A -85,B 0,C 180,E1 21077.238,E2 21077.238} C_VEL
LIN {X 0,Y 226.648,Z 805.023,A -85,B 0,C 180,E1 21083.701,E2 21083.701} C_VEL
LIN {X 0,Y 194.252,Z 851.334,A -85,B 0,C 180,E1 21094.884,E2 21094.884} C_VEL
LIN {X 0,Y 167.982,Z 885.296,A -85,B 0,C 180,E1 21112.423,E2 21112.423} C_VEL
LIN {X 0,Y 157.817,Z 903.636,A -85,B 0,C 180,E1 21132.878,E2 21132.878} C_VEL
LIN {X 0,Y 157.465,Z 908.588,A -85,B 0,C 180,E1 21147.236,E2 21147.236} C_VEL
LIN {X 0,Y 157.388,Z 906.112,A -85,B 0,C 180,E1 21163.946,E2 21163.946} C_VEL
LIN {X 0,Y 167.7,Z 889.058,A -85,B 0,C 180,E1 21187.604,E2 21187.604} C_VEL
LIN {X 0,Y 199.147,Z 855.642,A -85,B 0,C 180,E1 21206.948,E2 21206.948} C_VEL
LIN {X 0,Y 237.119,Z 811.759,A -85,B 0,C 180,E1 21218.117,E2 21218.117} C_VEL
LIN {X 0,Y 271.943,Z 758.309,A -85,B 0,C 180,E1 21224.699,E2 21224.699} C_VEL
LIN {X 0,Y 272.843,Z 745.169,A -85,B 0,C 180,E1 21232.072,E2 21232.072} C_VEL
LIN {X 0,Y 271.799,Z 744.55,A -85,B 0,C 180,E1 21238.462,E2 21238.462} C_VEL
LIN {X 0,Y 268.063,Z 753.98,A -85,B 0,C 180,E1 21243.922,E2 21243.922} C_VEL
LIN {X 0,Y 234.059,Z 799.865,A -85,B 0,C 180,E1 21250.701,E2 21250.701} C_VEL
LIN {X 0,Y 200.275,Z 832.909,A -85,B 0,C 180,E1 21261.404,E2 21261.404} C_VEL
LIN {X 0,Y 173.442,Z 853.249,A -85,B 0,C 180,E1 21277.156,E2 21277.156} C_VEL
LIN {X 0,Y 167.272,Z 857.076,A -85,B 0,C 180,E1 21283.607,E2 21283.607} C_VEL
LIN {X 0,Y 152.663,Z 861.565,A -85,B 0,C 180,E1 21295.13,E2 21295.13} C_VEL
LIN {X 0,Y 154.389,Z 856.178,A -85,B 0,C 180,E1 21318.085,E2 21318.085} C_VEL
LIN {X 0,Y 170.922,Z 837.299,A -85,B 0,C 180,E1 21337.656,E2 21337.656} C_VEL
LIN {X 0,Y 198.137,Z 804.521,A -85,B 0,C 180,E1 21351.936,E2 21351.936} C_VEL
LIN {X 0,Y 227.839,Z 758.822,A -85,B 0,C 180,E1 21361.079,E2 21361.079} C_VEL
LIN {X 0,Y 238.651,Z 736.231,A -85,B 0,C 180,E1 21363.959,E2 21363.959} C_VEL
LIN {X 0,Y 234.771,Z 711.357,A -85,B 0,C 180,E1 21374.811,E2 21374.811} C_VEL
LIN {X 0,Y 230.281,Z 694.734,A -85,B 0,C 180,E1 21388.392,E2 21388.392} C_VEL
LIN {X 0,Y 230.746,Z 692.005,A -85,B 0,C 180,E1 21402.484,E2 21402.484} C_VEL
LIN {X 0,Y 235.546,Z 700.457,A -85,B 0,C 180,E1 21413.643,E2 21413.643} C_VEL
LIN {X 0,Y 243.051,Z 725.523,A -85,B 0,C 180,E1 21426.202,E2 21426.202} C_VEL
LIN {X 0,Y 248.37,Z 755.705,A -85,B 0,C 180,E1 21436.122,E2 21436.122} C_VEL
LIN {X 0,Y 217.634,Z 810.779,A -85,B 0,C 180,E1 21443.137,E2 21443.137} C_VEL
LIN {X 0,Y 184.208,Z 855.645,A -85,B 0,C 180,E1 21455.139,E2 21455.139} C_VEL
LIN {X 0,Y 158.719,Z 887.089,A -85,B 0,C 180,E1 21473.459,E2 21473.459} C_VEL
LIN {X 0,Y 149.596,Z 903.828,A -85,B 0,C 180,E1 21495.306,E2 21495.306} C_VEL
LIN {X 0,Y 149.553,Z 907.526,A -85,B 0,C 180,E1 21512.906,E2 21512.906} C_VEL
LIN {X 0,Y 150.196,Z 902.219,A -85,B 0,C 180,E1 21530.706,E2 21530.706} C_VEL
LIN {X 0,Y 167.063,Z 881.625,A -85,B 0,C 180,E1 21554.743,E2 21554.743} C_VEL
LIN {X 0,Y 203.669,Z 845.394,A -85,B 0,C 180,E1 21572.222,E2 21572.222} C_VEL
LIN {X 0,Y 243.353,Z 799.126,A -85,B 0,C 180,E1 21581.82,E2 21581.82} C_VEL
LIN {X 0,Y 267.452,Z 762.253,A -85,B 0,C 180,E1 21586.023,E2 21586.023} C_VEL
LIN {X 0,Y 268.581,Z 752.198,A -85,B 0,C 180,E1 21591.945,E2 21591.945} C_VEL
LIN {X 0,Y 267.498,Z 751.544,A -85,B 0,C 180,E1 21598.437,E2 21598.437} C_VEL
LIN {X 0,Y 264.192,Z 758.436,A -85,B 0,C 180,E1 21602.578,E2 21602.578} C_VEL
LIN {X 0,Y 229.12,Z 803.183,A -85,B 0,C 180,E1 21609.319,E2 21609.319} C_VEL
LIN {X 0,Y 192.03,Z 836.968,A -85,B 0,C 180,E1 21620.915,E2 21620.915} C_VEL
LIN {X 0,Y 164.087,Z 856.222,A -85,B 0,C 180,E1 21638.181,E2 21638.181} C_VEL
LIN {X 0,Y 152.663,Z 861.565,A -85,B 0,C 180,E1 21655.13,E2 21655.13} C_VEL
LIN {X 0,Y 143.492,Z 861.414,A -85,B 0,C 180,E1 21668.453,E2 21668.453} C_VEL
LIN {X 0,Y 154.069,Z 849.075,A -85,B 0,C 180,E1 21690.057,E2 21690.057} C_VEL
LIN {X 0,Y 179.142,Z 821.997,A -85,B 0,C 180,E1 21707.885,E2 21707.885} C_VEL
LIN {X 0,Y 210.067,Z 781.835,A -85,B 0,C 180,E1 21719.186,E2 21719.186} C_VEL
LIN {X 0,Y 233.518,Z 739.141,A -85,B 0,C 180,E1 21725.587,E2 21725.587} C_VEL
LIN {X 0,Y 230.553,Z 716.538,A -85,B 0,C 180,E1 21736.204,E2 21736.204} C_VEL
LIN {X 0,Y 227.428,Z 702.569,A -85,B 0,C 180,E1 21747.948,E2 21747.948} C_VEL
LIN {X 0,Y 227.378,Z 698.628,A -85,B 0,C 180,E1 21758.396,E2 21758.396} C_VEL
LIN {X 0,Y 230.855,Z 704.776,A -85,B 0,C 180,E1 21770.472,E2 21770.472} C_VEL
LIN {X 0,Y 236.755,Z 723.392,A -85,B 0,C 180,E1 21782.06,E2 21782.06} C_VEL
LIN {X 0,Y 242.25,Z 754.756,A -85,B 0,C 180,E1 21793.602,E2 21793.602} C_VEL
LIN {X 0,Y 241.09,Z 762.572,A -85,B 0,C 180,E1 21795.29,E2 21795.29} C_VEL
LIN {X 0,Y 207.786,Z 817.363,A -85,B 0,C 180,E1 21802.769,E2 21802.769} C_VEL
LIN {X 0,Y 173.232,Z 860.665,A -85,B 0,C 180,E1 21815.871,E2 21815.871} C_VEL
LIN {X 0,Y 148.498,Z 889.844,A -85,B 0,C 180,E1 21835.799,E2 21835.799} C_VEL
LIN {X 0,Y 141.458,Z 903.74,A -85,B 0,C 180,E1 21857.608,E2 21857.608} C_VEL
LIN {X 0,Y 141.611,Z 906.269,A -85,B 0,C 180,E1 21873.069,E2 21873.069} C_VEL
LIN {X 0,Y 143.118,Z 899.759,A -85,B 0,C 180,E1 21894.313,E2 21894.313} C_VEL
LIN {X 0,Y 163.016,Z 878.801,A -85,B 0,C 180,E1 21918.131,E2 21918.131} C_VEL
LIN {X 0,Y 201.073,Z 843.312,A -85,B 0,C 180,E1 21934.732,E2 21934.732} C_VEL
LIN {X 0,Y 242.059,Z 797.013,A -85,B 0,C 180,E1 21943.924,E2 21943.924} C_VEL
LIN {X 0,Y 263.117,Z 765.875,A -85,B 0,C 180,E1 21947.556,E2 21947.556} C_VEL
LIN {X 0,Y 264.198,Z 756.907,A -85,B 0,C 180,E1 21955.122,E2 21955.122} C_VEL
LIN {X 0,Y 260.936,Z 762.135,A -85,B 0,C 180,E1 21961.125,E2 21961.125} C_VEL
LIN {X 0,Y 224.323,Z 806.41,A -85,B 0,C 180,E1 21967.862,E2 21967.862} C_VEL
LIN {X 0,Y 187.155,Z 838.423,A -85,B 0,C 180,E1 21979.015,E2 21979.015} C_VEL
LIN {X 0,Y 158.52,Z 856.946,A -85,B 0,C 180,E1 21995.544,E2 21995.544} C_VEL
LIN {X 0,Y 144.849,Z 862.932,A -85,B 0,C 180,E1 22014.819,E2 22014.819} C_VEL
LIN {X 0,Y 143.492,Z 861.414,A -85,B 0,C 180,E1 22028.453,E2 22028.453} C_VEL
LIN {X 0,Y 140.599,Z 856.635,A -85,B 0,C 180,E1 22042.657,E2 22042.657} C_VEL
LIN {X 0,Y 162.156,Z 835.026,A -85,B 0,C 180,E1 22063.533,E2 22063.533} C_VEL
LIN {X 0,Y 192.214,Z 800.864,A -85,B 0,C 180,E1 22077,E2 22077} C_VEL
LIN {X 0,Y 223.663,Z 753.271,A -85,B 0,C 180,E1 22085.477,E2 22085.477} C_VEL
LIN {X 0,Y 228.496,Z 743.133,A -85,B 0,C 180,E1 22086.903,E2 22086.903} C_VEL
LIN {X 0,Y 226.298,Z 721.513,A -85,B 0,C 180,E1 22097.796,E2 22097.796} C_VEL
LIN {X 0,Y 224.09,Z 709.228,A -85,B 0,C 180,E1 22109.404,E2 22109.404} C_VEL
LIN {X 0,Y 225.106,Z 706.981,A -85,B 0,C 180,E1 22122.27,E2 22122.27} C_VEL
LIN {X 0,Y 229.055,Z 715.276,A -85,B 0,C 180,E1 22133.272,E2 22133.272} C_VEL
LIN {X 0,Y 234.42,Z 739.083,A -85,B 0,C 180,E1 22145.499,E2 22145.499} C_VEL
LIN {X 0,Y 236.403,Z 763.445,A -85,B 0,C 180,E1 22153.743,E2 22153.743} C_VEL
LIN {X 0,Y 203.103,Z 816.576,A -85,B 0,C 180,E1 22160.934,E2 22160.934} C_VEL
LIN {X 0,Y 167.189,Z 859.857,A -85,B 0,C 180,E1 22174.077,E2 22174.077} C_VEL
LIN {X 0,Y 140.479,Z 889.587,A -85,B 0,C 180,E1 22195.446,E2 22195.446} C_VEL
LIN {X 0,Y 133.449,Z 903.372,A -85,B 0,C 180,E1 22220.176,E2 22220.176} C_VEL
LIN {X 0,Y 133.648,Z 905.004,A -85,B 0,C 180,E1 22233.252,E2 22233.252} C_VEL
LIN {X 0,Y 135.511,Z 898.674,A -85,B 0,C 180,E1 22255.535,E2 22255.535} C_VEL
LIN {X 0,Y 158.722,Z 876.729,A -85,B 0,C 180,E1 22281.158,E2 22281.158} C_VEL
LIN {X 0,Y 199.914,Z 840.326,A -85,B 0,C 180,E1 22297.557,E2 22297.557} C_VEL
LIN {X 0,Y 242.215,Z 793.609,A -85,B 0,C 180,E1 22306.185,E2 22306.185} C_VEL
LIN {X 0,Y 258.654,Z 770.144,A -85,B 0,C 180,E1 22308.931,E2 22308.931} C_VEL
LIN {X 0,Y 259.689,Z 763.609,A -85,B 0,C 180,E1 22315.037,E2 22315.037} C_VEL
LIN {X 0,Y 256.668,Z 767.424,A -85,B 0,C 180,E1 22319.817,E2 22319.817} C_VEL
LIN {X 0,Y 218.529,Z 810.689,A -85,B 0,C 180,E1 22326.563,E2 22326.563} C_VEL
LIN {X 0,Y 178.991,Z 842.354,A -85,B 0,C 180,E1 22338.379,E2 22338.379} C_VEL
LIN {X 0,Y 148.385,Z 860.143,A -85,B 0,C 180,E1 22357.222,E2 22357.222} C_VEL
LIN {X 0,Y 135.718,Z 864.127,A -85,B 0,C 180,E1 22379.794,E2 22379.794} C_VEL
LIN {X 0,Y 140.599,Z 856.635,A -85,B 0,C 180,E1 22402.657,E2 22402.657} C_VEL
LIN {X 0,Y 143.541,Z 847.637,A -85,B 0,C 180,E1 22416.51,E2 22416.51} C_VEL
LIN {X 0,Y 173.273,Z 818.115,A -85,B 0,C 180,E1 22433.92,E2 22433.92} C_VEL
LIN {X 0,Y 206.889,Z 775.384,A -85,B 0,C 180,E1 22444.326,E2 22444.326} C_VEL
LIN {X 0,Y 223.438,Z 746.392,A -85,B 0,C 180,E1 22448.554,E2 22448.554} C_VEL
LIN {X 0,Y 222.07,Z 726.596,A -85,B 0,C 180,E1 22459.441,E2 22459.441} C_VEL
LIN {X 0,Y 220.875,Z 716.741,A -85,B 0,C 180,E1 22469.187,E2 22469.187} C_VEL
LIN {X 0,Y 221.894,Z 714.291,A -85,B 0,C 180,E1 22482.005,E2 22482.005} C_VEL
LIN {X 0,Y 225.914,Z 724.155,A -85,B 0,C 180,E1 22494.146,E2 22494.146} C_VEL
LIN {X 0,Y 230.234,Z 749.267,A -85,B 0,C 180,E1 22506.548,E2 22506.548} C_VEL
LIN {X 0,Y 230.204,Z 767.23,A -85,B 0,C 180,E1 22512.417,E2 22512.417} C_VEL
LIN {X 0,Y 196.074,Z 818.968,A -85,B 0,C 180,E1 22519.686,E2 22519.686} C_VEL
LIN {X 0,Y 159.892,Z 860.437,A -85,B 0,C 180,E1 22532.851,E2 22532.851} C_VEL
LIN {X 0,Y 132.454,Z 889.284,A -85,B 0,C 180,E1 22555.047,E2 22555.047} C_VEL
LIN {X 0,Y 125.523,Z 902.029,A -85,B 0,C 180,E1 22579.549,E2 22579.549} C_VEL
LIN {X 0,Y 125.696,Z 903.742,A -85,B 0,C 180,E1 22593.458,E2 22593.458} C_VEL
LIN {X 0,Y 128.356,Z 897.145,A -85,B 0,C 180,E1 22617.859,E2 22617.859} C_VEL
LIN {X 0,Y 155.011,Z 874.515,A -85,B 0,C 180,E1 22644.49,E2 22644.49} C_VEL
LIN {X 0,Y 198.378,Z 838.186,A -85,B 0,C 180,E1 22660.197,E2 22660.197} C_VEL
LIN {X 0,Y 241.792,Z 791.509,A -85,B 0,C 180,E1 22668.293,E2 22668.293} C_VEL
LIN {X 0,Y 254.061,Z 774.702,A -85,B 0,C 180,E1 22670.24,E2 22670.24} C_VEL
LIN {X 0,Y 254.915,Z 770.146,A -85,B 0,C 180,E1 22674.944,E2 22674.944} C_VEL
LIN {X 0,Y 251.805,Z 773.643,A -85,B 0,C 180,E1 22678.544,E2 22678.544} C_VEL
LIN {X 0,Y 211.462,Z 816.165,A -85,B 0,C 180,E1 22685.522,E2 22685.522} C_VEL
LIN {X 0,Y 171.084,Z 845.883,A -85,B 0,C 180,E1 22697.552,E2 22697.552} C_VEL
LIN {X 0,Y 140.624,Z 861.936,A -85,B 0,C 180,E1 22716.537,E2 22716.537} C_VEL
LIN {X 0,Y 127.418,Z 864.858,A -85,B 0,C 180,E1 22743.528,E2 22743.528} C_VEL
LIN {X 0,Y 136.522,Z 854.403,A -85,B 0,C 180,E1 22768.771,E2 22768.771} C_VEL
LIN {X 0,Y 143.541,Z 847.637,A -85,B 0,C 180,E1 22776.51,E2 22776.51} C_VEL
LIN {X 0,Y 152.709,Z 834.431,A -85,B 0,C 180,E1 22788.779,E2 22788.779} C_VEL
LIN {X 0,Y 186.383,Z 798.496,A -85,B 0,C 180,E1 22801.956,E2 22801.956} C_VEL
LIN {X 0,Y 218.439,Z 751.229,A -85,B 0,C 180,E1 22809.606,E2 22809.606} C_VEL
LIN {X 0,Y 217.832,Z 731.638,A -85,B 0,C 180,E1 22821.154,E2 22821.154} C_VEL
LIN {X 0,Y 217.188,Z 722.454,A -85,B 0,C 180,E1 22832.915,E2 22832.915} C_VEL
LIN {X 0,Y 219.607,Z 723.314,A -85,B 0,C 180,E1 22845.932,E2 22845.932} C_VEL
LIN {X 0,Y 222.682,Z 734.879,A -85,B 0,C 180,E1 22856.149,E2 22856.149} C_VEL
LIN {X 0,Y 225.697,Z 761.038,A -85,B 0,C 180,E1 22868.258,E2 22868.258} C_VEL
LIN {X 0,Y 224.182,Z 770.777,A -85,B 0,C 180,E1 22871.022,E2 22871.022} C_VEL
LIN {X 0,Y 188.535,Z 822.116,A -85,B 0,C 180,E1 22878.516,E2 22878.516} C_VEL
LIN {X 0,Y 150.601,Z 863.11,A -85,B 0,C 180,E1 22892.579,E2 22892.579} C_VEL
LIN {X 0,Y 123.258,Z 890.283,A -85,B 0,C 180,E1 22916.353,E2 22916.353} C_VEL
LIN {X 0,Y 117.611,Z 900.673,A -85,B 0,C 180,E1 22938.837,E2 22938.837} C_VEL
LIN {X 0,Y 117.722,Z 902.471,A -85,B 0,C 180,E1 22953.692,E2 22953.692} C_VEL
LIN {X 0,Y 121.027,Z 895.958,A -85,B 0,C 180,E1 22979.709,E2 22979.709} C_VEL
LIN {X 0,Y 149.267,Z 874.23,A -85,B 0,C 180,E1 23006.63,E2 23006.63} C_VEL
LIN {X 0,Y 193.964,Z 839.014,A -85,B 0,C 180,E1 23022.129,E2 23022.129} C_VEL
LIN {X 0,Y 238.816,Z 793.017,A -85,B 0,C 180,E1 23030.028,E2 23030.028} C_VEL
LIN {X 0,Y 248.723,Z 780.438,A -85,B 0,C 180,E1 23031.297,E2 23031.297} C_VEL
LIN {X 0,Y 249.996,Z 776.621,A -85,B 0,C 180,E1 23034.845,E2 23034.845} C_VEL
LIN {X 0,Y 247.216,Z 779.375,A -85,B 0,C 180,E1 23037.219,E2 23037.219} C_VEL
LIN {X 0,Y 205.411,Z 820.603,A -85,B 0,C 180,E1 23044.204,E2 23044.204} C_VEL
LIN {X 0,Y 162.726,Z 849.64,A -85,B 0,C 180,E1 23056.846,E2 23056.846} C_VEL
LIN {X 0,Y 131.777,Z 864.166,A -85,B 0,C 180,E1 23076.885,E2 23076.885} C_VEL
LIN {X 0,Y 119.535,Z 866.037,A -85,B 0,C 180,E1 23103.623,E2 23103.623} C_VEL
LIN {X 0,Y 130.503,Z 854.359,A -85,B 0,C 180,E1 23131.703,E2 23131.703} C_VEL
LIN {X 0,Y 152.709,Z 834.431,A -85,B 0,C 180,E1 23148.779,E2 23148.779} C_VEL
LIN {X 0,Y 165.625,Z 817.434,A -85,B 0,C 180,E1 23158.999,E2 23158.999} C_VEL
LIN {X 0,Y 201.505,Z 773.919,A -85,B 0,C 180,E1 23168.759,E2 23168.759} C_VEL
LIN {X 0,Y 213.575,Z 754.067,A -85,B 0,C 180,E1 23171.659,E2 23171.659} C_VEL
LIN {X 0,Y 213.72,Z 736.89,A -85,B 0,C 180,E1 23182.796,E2 23182.796} C_VEL
LIN {X 0,Y 213.609,Z 729.778,A -85,B 0,C 180,E1 23192.63,E2 23192.63} C_VEL
LIN {X 0,Y 215.958,Z 730.39,A -85,B 0,C 180,E1 23205.689,E2 23205.689} C_VEL
LIN {X 0,Y 218.52,Z 742.071,A -85,B 0,C 180,E1 23216.075,E2 23216.075} C_VEL
LIN {X 0,Y 220.312,Z 767.011,A -85,B 0,C 180,E1 23227.808,E2 23227.808} C_VEL
LIN {X 0,Y 218.073,Z 774.569,A -85,B 0,C 180,E1 23229.599,E2 23229.599} C_VEL
LIN {X 0,Y 180.829,Z 825.328,A -85,B 0,C 180,E1 23237.325,E2 23237.325} C_VEL
LIN {X 0,Y 142.489,Z 864.304,A -85,B 0,C 180,E1 23251.576,E2 23251.576} C_VEL
LIN {X 0,Y 115.329,Z 889.763,A -85,B 0,C 180,E1 23275.753,E2 23275.753} C_VEL
LIN {X 0,Y 109.707,Z 899.317,A -85,B 0,C 180,E1 23298.021,E2 23298.021} C_VEL
LIN {X 0,Y 109.744,Z 901.202,A -85,B 0,C 180,E1 23313.961,E2 23313.961} C_VEL
LIN {X 0,Y 114.168,Z 894.522,A -85,B 0,C 180,E1 23342.399,E2 23342.399} C_VEL
LIN {X 0,Y 147.751,Z 871.274,A -85,B 0,C 180,E1 23370.806,E2 23370.806} C_VEL
LIN {X 0,Y 195.959,Z 834.606,A -85,B 0,C 180,E1 23385.46,E2 23385.46} C_VEL
LIN {X 0,Y 243.009,Z 786.327,A -85,B 0,C 180,E1 23392.63,E2 23392.63} C_VEL
LIN {X 0,Y 244.875,Z 782.95,A -85,B 0,C 180,E1 23394.736,E2 23394.736} C_VEL
LIN {X 0,Y 240.17,Z 787.838,A -85,B 0,C 180,E1 23396.17,E2 23396.17} C_VEL
LIN {X 0,Y 196.269,Z 827.324,A -85,B 0,C 180,E1 23403.483,E2 23403.483} C_VEL
LIN {X 0,Y 151.127,Z 854.776,A -85,B 0,C 180,E1 23417.468,E2 23417.468} C_VEL
LIN {X 0,Y 123.292,Z 866.085,A -85,B 0,C 180,E1 23436.871,E2 23436.871} C_VEL
LIN {X 0,Y 111.661,Z 867.385,A -85,B 0,C 180,E1 23462.328,E2 23462.328} C_VEL
LIN {X 0,Y 122.229,Z 856.452,A -85,B 0,C 180,E1 23491.819,E2 23491.819} C_VEL
LIN {X 0,Y 151.009,Z 831.752,A -85,B 0,C 180,E1 23512.92,E2 23512.92} C_VEL
LIN {X 0,Y 165.625,Z 817.434,A -85,B 0,C 180,E1 23518.999,E2 23518.999} C_VEL
LIN {X 0,Y 181.219,Z 796.628,A -85,B 0,C 180,E1 23526.998,E2 23526.998} C_VEL
LIN {X 0,Y 208.587,Z 758.664,A -85,B 0,C 180,E1 23532.89,E2 23532.89} C_VEL
LIN {X 0,Y 209.482,Z 742.72,A -85,B 0,C 180,E1 23543.974,E2 23543.974} C_VEL
LIN {X 0,Y 210.285,Z 735.649,A -85,B 0,C 180,E1 23556.539,E2 23556.539} C_VEL
LIN {X 0,Y 213.117,Z 740.587,A -85,B 0,C 180,E1 23569.671,E2 23569.671} C_VEL
LIN {X 0,Y 214.862,Z 759.349,A -85,B 0,C 180,E1 23581.44,E2 23581.44} C_VEL
LIN {X 0,Y 213.511,Z 775.789,A -85,B 0,C 180,E1 23587.862,E2 23587.862} C_VEL
LIN {X 0,Y 176.728,Z 824.412,A -85,B 0,C 180,E1 23595.094,E2 23595.094} C_VEL
LIN {X 0,Y 136.544,Z 863.646,A -85,B 0,C 180,E1 23609.377,E2 23609.377} C_VEL
LIN {X 0,Y 107.183,Z 889.418,A -85,B 0,C 180,E1 23635.501,E2 23635.501} C_VEL
LIN {X 0,Y 101.789,Z 897.94,A -85,B 0,C 180,E1 23657.074,E2 23657.074} C_VEL
LIN {X 0,Y 101.757,Z 899.925,A -85,B 0,C 180,E1 23674.272,E2 23674.272} C_VEL
LIN {X 0,Y 107.037,Z 893.456,A -85,B 0,C 180,E1 23704.544,E2 23704.544} C_VEL
LIN {X 0,Y 143.797,Z 870.333,A -85,B 0,C 180,E1 23733.763,E2 23733.763} C_VEL
LIN {X 0,Y 194.005,Z 834.035,A -85,B 0,C 180,E1 23747.883,E2 23747.883} C_VEL
LIN {X 0,Y 238.345,Z 790.542,A -85,B 0,C 180,E1 23754.423,E2 23754.423} C_VEL
LIN {X 0,Y 192.524,Z 829.952,A -85,B 0,C 180,E1 23761.545,E2 23761.545} C_VEL
LIN {X 0,Y 146.085,Z 856.549,A -85,B 0,C 180,E1 23775.164,E2 23775.164} C_VEL
LIN {X 0,Y 114.975,Z 867.883,A -85,B 0,C 180,E1 23796.6,E2 23796.6} C_VEL
LIN {X 0,Y 103.861,Z 867.489,A -85,B 0,C 180,E1 23828.579,E2 23828.579} C_VEL
LIN {X 0,Y 118.445,Z 854.813,A -85,B 0,C 180,E1 23857.364,E2 23857.364} C_VEL
LIN {X 0,Y 151.726,Z 827.274,A -85,B 0,C 180,E1 23877.838,E2 23877.838} C_VEL
LIN {X 0,Y 181.219,Z 796.628,A -85,B 0,C 180,E1 23886.998,E2 23886.998} C_VEL
LIN {X 0,Y 196.999,Z 772.624,A -85,B 0,C 180,E1 23893.329,E2 23893.329} C_VEL
LIN {X 0,Y 203.856,Z 761.788,A -85,B 0,C 180,E1 23895.009,E2 23895.009} C_VEL
LIN {X 0,Y 205.336,Z 747.558,A -85,B 0,C 180,E1 23906.257,E2 23906.257} C_VEL
LIN {X 0,Y 207.157,Z 742.699,A -85,B 0,C 180,E1 23920.676,E2 23920.676} C_VEL
LIN {X 0,Y 209.302,Z 749.788,A -85,B 0,C 180,E1 23931.586,E2 23931.586} C_VEL
LIN {X 0,Y 209.735,Z 770.941,A -85,B 0,C 180,E1 23943.549,E2 23943.549} C_VEL
LIN {X 0,Y 208.306,Z 778.289,A -85,B 0,C 180,E1 23946.191,E2 23946.191} C_VEL
LIN {X 0,Y 169.355,Z 827.268,A -85,B 0,C 180,E1 23953.601,E2 23953.601} C_VEL
LIN {X 0,Y 127.529,Z 865.663,A -85,B 0,C 180,E1 23968.642,E2 23968.642} C_VEL
LIN {X 0,Y 98.08,Z 890.061,A -85,B 0,C 180,E1 23997.207,E2 23997.207} C_VEL
LIN {X 0,Y 93.811,Z 898.197,A -85,B 0,C 180,E1 24025.357,E2 24025.357} C_VEL
LIN {X 0,Y 93.565,Z 897.933,A -85,B 0,C 180,E1 24044.076,E2 24044.076} C_VEL
LIN {X 0,Y 109.994,Z 886.53,A -85,B 0,C 180,E1 24079.353,E2 24079.353} C_VEL
LIN {X 0,Y 157.388,Z 858.795,A -85,B 0,C 180,E1 24102.639,E2 24102.639} C_VEL
LIN {X 0,Y 209.831,Z 818.752,A -85,B 0,C 180,E1 24112.902,E2 24112.902} C_VEL
LIN {X 0,Y 221.043,Z 808.078,A -85,B 0,C 180,E1 24114.522,E2 24114.522} C_VEL
LIN {X 0,Y 173.294,Z 842.292,A -85,B 0,C 180,E1 24122.869,E2 24122.869} C_VEL
LIN {X 0,Y 128.689,Z 863.17,A -85,B 0,C 180,E1 24138.664,E2 24138.664} C_VEL
LIN {X 0,Y 99.814,Z 870.586,A -85,B 0,C 180,E1 24166.836,E2 24166.836} C_VEL
LIN {X 0,Y 99.741,Z 864.843,A -85,B 0,C 180,E1 24202.504,E2 24202.504} C_VEL
LIN {X 0,Y 124.724,Z 846.292,A -85,B 0,C 180,E1 24229.551,E2 24229.551} C_VEL
LIN {X 0,Y 163.013,Z 813.017,A -85,B 0,C 180,E1 24245.582,E2 24245.582} C_VEL
LIN {X 0,Y 196.999,Z 772.624,A -85,B 0,C 180,E1 24253.329,E2 24253.329} C_VEL
LIN {X 0,Y 199.858,Z 764.85,A -85,B 0,C 180,E1 24256.764,E2 24256.764} C_VEL
LIN {X 0,Y 199.775,Z 761.818,A -85,B 0,C 180,E1 24259.468,E2 24259.468} C_VEL
LIN {X 0,Y 201.287,Z 751.674,A -85,B 0,C 180,E1 24270.575,E2 24270.575} C_VEL
LIN {X 0,Y 202.911,Z 749.522,A -85,B 0,C 180,E1 24280.255,E2 24280.255} C_VEL
LIN {X 0,Y 204.863,Z 756.622,A -85,B 0,C 180,E1 24291.402,E2 24291.402} C_VEL
LIN {X 0,Y 204.167,Z 778.041,A -85,B 0,C 180,E1 24303.646,E2 24303.646} C_VEL
LIN {X 0,Y 167.252,Z 824.682,A -85,B 0,C 180,E1 24310.802,E2 24310.802} C_VEL
LIN {X 0,Y 125.086,Z 862.449,A -85,B 0,C 180,E1 24324.503,E2 24324.503} C_VEL
LIN {X 0,Y 92.458,Z 887.327,A -85,B 0,C 180,E1 24352.007,E2 24352.007} C_VEL
LIN {X 0,Y 85.831,Z 896.873,A -85,B 0,C 180,E1 24384.924,E2 24384.924} C_VEL
LIN {X 0,Y 85.655,Z 896.672,A -85,B 0,C 180,E1 24405.407,E2 24405.407} C_VEL
LIN {X 0,Y 104.639,Z 885.424,A -85,B 0,C 180,E1 24442.898,E2 24442.898} C_VEL
LIN {X 0,Y 155.078,Z 858.037,A -85,B 0,C 180,E1 24465.662,E2 24465.662} C_VEL
LIN {X 0,Y 203.442,Z 823.206,A -85,B 0,C 180,E1 24474.476,E2 24474.476} C_VEL
LIN {X 0,Y 151.386,Z 853.8,A -85,B 0,C 180,E1 24485.293,E2 24485.293} C_VEL
LIN {X 0,Y 109.072,Z 869.013,A -85,B 0,C 180,E1 24505.273,E2 24505.273} C_VEL
LIN {X 0,Y 89.291,Z 871.726,A -85,B 0,C 180,E1 24533.505,E2 24533.505} C_VEL
LIN {X 0,Y 97.003,Z 862.514,A -85,B 0,C 180,E1 24572.245,E2 24572.245} C_VEL
LIN {X 0,Y 129.6,Z 839.503,A -85,B 0,C 180,E1 24597.529,E2 24597.529} C_VEL
LIN {X 0,Y 169,Z 803.899,A -85,B 0,C 180,E1 24610.46,E2 24610.46} C_VEL
LIN {X 0,Y 199.023,Z 766.349,A -85,B 0,C 180,E1 24616.418,E2 24616.418} C_VEL
LIN {X 0,Y 199.775,Z 761.818,A -85,B 0,C 180,E1 24619.468,E2 24619.468} C_VEL
LIN {X 0,Y 196.708,Z 758.88,A -85,B 0,C 180,E1 24629.761,E2 24629.761} C_VEL
LIN {X 0,Y 198.94,Z 756.958,A -85,B 0,C 180,E1 24642.466,E2 24642.466} C_VEL
LIN {X 0,Y 200.074,Z 764.727,A -85,B 0,C 180,E1 24652.292,E2 24652.292} C_VEL
LIN {X 0,Y 198.787,Z 782.122,A -85,B 0,C 180,E1 24662.376,E2 24662.376} C_VEL
LIN {X 0,Y 157.561,Z 830.003,A -85,B 0,C 180,E1 24669.63,E2 24669.63} C_VEL
LIN {X 0,Y 114.64,Z 865.54,A -85,B 0,C 180,E1 24684.118,E2 24684.118} C_VEL
LIN {X 0,Y 82.241,Z 888.755,A -85,B 0,C 180,E1 24715.741,E2 24715.741} C_VEL
LIN {X 0,Y 77.851,Z 895.551,A -85,B 0,C 180,E1 24744.402,E2 24744.402} C_VEL
LIN {X 0,Y 77.79,Z 895.41,A -85,B 0,C 180,E1 24767.009,E2 24767.009} C_VEL
LIN {X 0,Y 99.724,Z 884.318,A -85,B 0,C 180,E1 24806.812,E2 24806.812} C_VEL
LIN {X 0,Y 153.196,Z 857.324,A -85,B 0,C 180,E1 24828.74,E2 24828.74} C_VEL
LIN {X 0,Y 185.891,Z 835.968,A -85,B 0,C 180,E1 24834.708,E2 24834.708} C_VEL
LIN {X 0,Y 133.505,Z 861.464,A -85,B 0,C 180,E1 24846.949,E2 24846.949} C_VEL
LIN {X 0,Y 95.489,Z 872.064,A -85,B 0,C 180,E1 24869.074,E2 24869.074} C_VEL
LIN {X 0,Y 80.132,Z 870.981,A -85,B 0,C 180,E1 24909.395,E2 24909.395} C_VEL
LIN {X 0,Y 99.614,Z 857.407,A -85,B 0,C 180,E1 24945.183,E2 24945.183} C_VEL
LIN {X 0,Y 139.051,Z 829.27,A -85,B 0,C 180,E1 24965.919,E2 24965.919} C_VEL
LIN {X 0,Y 180.981,Z 787.67,A -85,B 0,C 180,E1 24975.933,E2 24975.933} C_VEL
LIN {X 0,Y 194.291,Z 770.171,A -85,B 0,C 180,E1 24978.308,E2 24978.308} C_VEL
LIN {X 0,Y 196.708,Z 758.88,A -85,B 0,C 180,E1 24989.761,E2 24989.761} C_VEL
LIN {X 0,Y 193.964,Z 763.199,A -85,B 0,C 180,E1 25000.132,E2 25000.132} C_VEL
LIN {X 0,Y 195.358,Z 768.692,A -85,B 0,C 180,E1 25010.122,E2 25010.122} C_VEL
LIN {X 0,Y 193.6,Z 784.539,A -85,B 0,C 180,E1 25020.235,E2 25020.235} C_VEL
LIN {X 0,Y 151.192,Z 831.938,A -85,B 0,C 180,E1 25027.605,E2 25027.605} C_VEL
LIN {X 0,Y 104.812,Z 867.856,A -85,B 0,C 180,E1 25043.341,E2 25043.341} C_VEL
LIN {X 0,Y 72.981,Z 889.233,A -85,B 0,C 180,E1 25078.672,E2 25078.672} C_VEL
LIN {X 0,Y 69.86,Z 894.217,A -85,B 0,C 180,E1 25103.759,E2 25103.759} C_VEL
LIN {X 0,Y 69.996,Z 894.152,A -85,B 0,C 180,E1 25128.972,E2 25128.972} C_VEL
LIN {X 0,Y 95.335,Z 883.231,A -85,B 0,C 180,E1 25171.092,E2 25171.092} C_VEL
LIN {X 0,Y 151.018,Z 857.016,A -85,B 0,C 180,E1 25191.724,E2 25191.724} C_VEL
LIN {X 0,Y 166.438,Z 847.753,A -85,B 0,C 180,E1 25195.246,E2 25195.246} C_VEL
LIN {X 0,Y 115.349,Z 867.769,A -85,B 0,C 180,E1 25209.378,E2 25209.378} C_VEL
LIN {X 0,Y 82.281,Z 874.305,A -85,B 0,C 180,E1 25233.916,E2 25233.916} C_VEL
LIN {X 0,Y 73.719,Z 870.524,A -85,B 0,C 180,E1 25278.126,E2 25278.126} C_VEL
LIN {X 0,Y 101.739,Z 853.457,A -85,B 0,C 180,E1 25314.221,E2 25314.221} C_VEL
LIN {X 0,Y 144.855,Z 822.163,A -85,B 0,C 180,E1 25331.527,E2 25331.527} C_VEL
LIN {X 0,Y 186.689,Z 778.208,A -85,B 0,C 180,E1 25339.649,E2 25339.649} C_VEL
LIN {X 0,Y 189.991,Z 772.843,A -85,B 0,C 180,E1 25341.342,E2 25341.342} C_VEL
LIN {X 0,Y 192.281,Z 764.668,A -85,B 0,C 180,E1 25351.623,E2 25351.623} C_VEL
LIN {X 0,Y 193.964,Z 763.199,A -85,B 0,C 180,E1 25360.132,E2 25360.132} C_VEL
LIN {X 0,Y 190.319,Z 775.442,A -85,B 0,C 180,E1 25370.153,E2 25370.153} C_VEL
LIN {X 0,Y 187.162,Z 789.766,A -85,B 0,C 180,E1 25378.808,E2 25378.808} C_VEL
LIN {X 0,Y 142.24,Z 836.134,A -85,B 0,C 180,E1 25385.94,E2 25385.94} C_VEL
LIN {X 0,Y 94.539,Z 870.21,A -85,B 0,C 180,E1 25402.636,E2 25402.636} C_VEL
LIN {X 0,Y 63.989,Z 889.387,A -85,B 0,C 180,E1 25441.679,E2 25441.679} C_VEL
LIN {X 0,Y 61.902,Z 892.869,A -85,B 0,C 180,E1 25462.953,E2 25462.953} C_VEL
LIN {X 0,Y 62.283,Z 892.89,A -85,B 0,C 180,E1 25491.43,E2 25491.43} C_VEL
LIN {X 0,Y 94.454,Z 881.132,A -85,B 0,C 180,E1 25537.479,E2 25537.479} C_VEL
LIN {X 0,Y 149.654,Z 856.376,A -85,B 0,C 180,E1 25555.362,E2 25555.362} C_VEL
LIN {X 0,Y 100.464,Z 871.983,A -85,B 0,C 180,E1 25570.959,E2 25570.959} C_VEL
LIN {X 0,Y 69.661,Z 875.74,A -85,B 0,C 180,E1 25600.328,E2 25600.328} C_VEL
LIN {X 0,Y 70.845,Z 868.572,A -85,B 0,C 180,E1 25651.701,E2 25651.701} C_VEL
LIN {X 0,Y 107.729,Z 847.625,A -85,B 0,C 180,E1 25683.385,E2 25683.385} C_VEL
LIN {X 0,Y 153.294,Z 812.835,A -85,B 0,C 180,E1 25696.897,E2 25696.897} C_VEL
LIN {X 0,Y 184.968,Z 778.336,A -85,B 0,C 180,E1 25702.257,E2 25702.257} C_VEL
LIN {X 0,Y 187.873,Z 770.501,A -85,B 0,C 180,E1 25713.537,E2 25713.537} C_VEL
LIN {X 0,Y 190.387,Z 771.563,A -85,B 0,C 180,E1 25725.965,E2 25725.965} C_VEL
LIN {X 0,Y 190.319,Z 775.442,A -85,B 0,C 180,E1 25730.153,E2 25730.153} C_VEL
LIN {X 0,Y 183.521,Z 789.741,A -85,B 0,C 180,E1 25735.683,E2 25735.683} C_VEL
LIN {X 0,Y 177.349,Z 798.178,A -85,B 0,C 180,E1 25737.201,E2 25737.201} C_VEL
LIN {X 0,Y 129.486,Z 843.094,A -85,B 0,C 180,E1 25744.987,E2 25744.987} C_VEL
LIN {X 0,Y 82.374,Z 873.408,A -85,B 0,C 180,E1 25763.067,E2 25763.067} C_VEL
LIN {X 0,Y 55.175,Z 889.316,A -85,B 0,C 180,E1 25805.627,E2 25805.627} C_VEL
LIN {X 0,Y 53.79,Z 892.223,A -85,B 0,C 180,E1 25838.102,E2 25838.102} C_VEL
LIN {X 0,Y 76.617,Z 884.881,A -85,B 0,C 180,E1 25893.025,E2 25893.025} C_VEL
LIN {X 0,Y 132.375,Z 863.951,A -85,B 0,C 180,E1 25915.428,E2 25915.428} C_VEL
LIN {X 0,Y 80.193,Z 876.056,A -85,B 0,C 180,E1 25936.699,E2 25936.699} C_VEL
LIN {X 0,Y 56.451,Z 874.319,A -85,B 0,C 180,E1 25991.018,E2 25991.018} C_VEL
LIN {X 0,Y 84.08,Z 859.392,A -85,B 0,C 180,E1 26036.827,E2 26036.827} C_VEL
LIN {X 0,Y 130.304,Z 830.494,A -85,B 0,C 180,E1 26055.559,E2 26055.559} C_VEL
LIN {X 0,Y 175.763,Z 788.103,A -85,B 0,C 180,E1 26063.521,E2 26063.521} C_VEL
LIN {X 0,Y 180.583,Z 781.878,A -85,B 0,C 180,E1 26065.027,E2 26065.027} C_VEL
LIN {X 0,Y 183.965,Z 776.023,A -85,B 0,C 180,E1 26078.122,E2 26078.122} C_VEL
LIN {X 0,Y 185.416,Z 779.655,A -85,B 0,C 180,E1 26088.107,E2 26088.107} C_VEL
LIN {X 0,Y 183.521,Z 789.741,A -85,B 0,C 180,E1 26095.683,E2 26095.683} C_VEL
LIN {X 0,Y 176.884,Z 797.634,A -85,B 0,C 180,E1 26096.304,E2 26096.304} C_VEL
LIN {X 0,Y 166.709,Z 806.865,A -85,B 0,C 180,E1 26095.594,E2 26095.594} C_VEL
LIN {X 0,Y 117.973,Z 848.477,A -85,B 0,C 180,E1 26103.545,E2 26103.545} C_VEL
LIN {X 0,Y 68.435,Z 877.047,A -85,B 0,C 180,E1 26125.225,E2 26125.225} C_VEL
LIN {X 0,Y 46.032,Z 890.06,A -85,B 0,C 180,E1 26180.504,E2 26180.504} C_VEL
LIN {X 0,Y 47.328,Z 890.357,A -85,B 0,C 180,E1 26218.738,E2 26218.738} C_VEL
LIN {X 0,Y 92.782,Z 878.021,A -85,B 0,C 180,E1 26268.892,E2 26268.892} C_VEL
LIN {X 0,Y 114.136,Z 870.406,A -85,B 0,C 180,E1 26275.65,E2 26275.65} C_VEL
LIN {X 0,Y 64.979,Z 878.239,A -85,B 0,C 180,E1 26300.77,E2 26300.77} C_VEL
LIN {X 0,Y 50.094,Z 874.152,A -85,B 0,C 180,E1 26361.296,E2 26361.296} C_VEL
LIN {X 0,Y 85.13,Z 857.423,A -85,B 0,C 180,E1 26404.631,E2 26404.631} C_VEL
LIN {X 0,Y 133.548,Z 826.858,A -85,B 0,C 180,E1 26420.091,E2 26420.091} C_VEL
LIN {X 0,Y 175.595,Z 787.071,A -85,B 0,C 180,E1 26426.291,E2 26426.291} C_VEL
LIN {X 0,Y 178.703,Z 782.474,A -85,B 0,C 180,E1 26437.443,E2 26437.443} C_VEL
LIN {X 0,Y 180.222,Z 785.724,A -85,B 0,C 180,E1 26447.759,E2 26447.759} C_VEL
LIN {X 0,Y 177.502,Z 794.924,A -85,B 0,C 180,E1 26454.503,E2 26454.503} C_VEL
LIN {X 0,Y 166.709,Z 806.865,A -85,B 0,C 180,E1 26455.594,E2 26455.594} C_VEL
LIN {X 0,Y 139.436,Z 829.638,A -85,B 0,C 180,E1 26455.841,E2 26455.841} C_VEL
LIN {X 0,Y 87.432,Z 864.324,A -85,B 0,C 180,E1 26467.267,E2 26467.267} C_VEL
LIN {X 0,Y 43.252,Z 884.918,A -85,B 0,C 180,E1 26507.2,E2 26507.2} C_VEL
LIN {X 0,Y 38.103,Z 888.631,A -85,B 0,C 180,E1 26538.503,E2 26538.503} C_VEL
LIN {X 0,Y 40.289,Z 889.031,A -85,B 0,C 180,E1 26584.39,E2 26584.39} C_VEL
LIN {X 0,Y 90.638,Z 877.258,A -85,B 0,C 180,E1 26633.85,E2 26633.85} C_VEL
LIN {X 0,Y 97.052,Z 875.322,A -85,B 0,C 180,E1 26635.689,E2 26635.689} C_VEL
LIN {X 0,Y 46.119,Z 879.34,A -85,B 0,C 180,E1 26674.668,E2 26674.668} C_VEL
LIN {X 0,Y 55.206,Z 869.687,A -85,B 0,C 180,E1 26750.104,E2 26750.104} C_VEL
LIN {X 0,Y 104.353,Z 845.845,A -85,B 0,C 180,E1 26777.458,E2 26777.458} C_VEL
LIN {X 0,Y 152.979,Z 809.618,A -85,B 0,C 180,E1 26786.462,E2 26786.462} C_VEL
LIN {X 0,Y 170.992,Z 791.369,A -85,B 0,C 180,E1 26788.886,E2 26788.886} C_VEL
LIN {X 0,Y 174.48,Z 788.886,A -85,B 0,C 180,E1 26802.185,E2 26802.185} C_VEL
LIN {X 0,Y 173.5,Z 796.155,A -85,B 0,C 180,E1 26811.292,E2 26811.292} C_VEL
LIN {X 0,Y 164.344,Z 806.696,A -85,B 0,C 180,E1 26812.955,E2 26812.955} C_VEL
LIN {X 0,Y 139.436,Z 829.638,A -85,B 0,C 180,E1 26815.841,E2 26815.841} C_VEL
LIN {X 0,Y 109.653,Z 848.923,A -85,B 0,C 180,E1 26816.579,E2 26816.579} C_VEL
LIN {X 0,Y 55.323,Z 876.494,A -85,B 0,C 180,E1 26836.224,E2 26836.224} C_VEL
LIN {X 0,Y 30.214,Z 887.199,A -85,B 0,C 180,E1 26895.442,E2 26895.442} C_VEL
LIN {X 0,Y 33.779,Z 887.69,A -85,B 0,C 180,E1 26952.35,E2 26952.35} C_VEL
LIN {X 0,Y 78.71,Z 879.231,A -85,B 0,C 180,E1 26996.145,E2 26996.145} C_VEL
LIN {X 0,Y 33.78,Z 879.52,A -85,B 0,C 180,E1 27047.651,E2 27047.651} C_VEL
LIN {X 0,Y 59.888,Z 866.784,A -85,B 0,C 180,E1 27125.149,E2 27125.149} C_VEL
LIN {X 0,Y 112.596,Z 840.182,A -85,B 0,C 180,E1 27143.971,E2 27143.971} C_VEL
LIN {X 0,Y 161.469,Z 801,A -85,B 0,C 180,E1 27150.386,E2 27150.386} C_VEL
LIN {X 0,Y 165.291,Z 797.116,A -85,B 0,C 180,E1 27150.719,E2 27150.719} C_VEL
LIN {X 0,Y 168.918,Z 794.823,A -85,B 0,C 180,E1 27161.578,E2 27161.578} C_VEL
LIN {X 0,Y 168.22,Z 800.046,A -85,B 0,C 180,E1 27169.482,E2 27169.482} C_VEL
LIN {X 0,Y 119.992,Z 842.031,A -85,B 0,C 180,E1 27174.87,E2 27174.87} C_VEL
LIN {X 0,Y 109.653,Z 848.923,A -85,B 0,C 180,E1 27176.579,E2 27176.579} C_VEL
LIN {X 0,Y 77.729,Z 864.405,A -85,B 0,C 180,E1 27178.115,E2 27178.115} C_VEL
LIN {X 0,Y 28.523,Z 883.177,A -85,B 0,C 180,E1 27217.034,E2 27217.034} C_VEL
LIN {X 0,Y 22.473,Z 885.753,A -85,B 0,C 180,E1 27250.249,E2 27250.249} C_VEL
LIN {X 0,Y 28.217,Z 886.354,A -85,B 0,C 180,E1 27323.751,E2 27323.751} C_VEL
LIN {X 0,Y 59.089,Z 882.034,A -85,B 0,C 180,E1 27357.025,E2 27357.025} C_VEL
LIN {X 0,Y 26.844,Z 877.713,A -85,B 0,C 180,E1 27450.015,E2 27450.015} C_VEL
LIN {X 0,Y 74.346,Z 860.384,A -85,B 0,C 180,E1 27499.954,E2 27499.954} C_VEL
LIN {X 0,Y 129.105,Z 828.701,A -85,B 0,C 180,E1 27510.38,E2 27510.38} C_VEL
LIN {X 0,Y 161.136,Z 801.247,A -85,B 0,C 180,E1 27513.472,E2 27513.472} C_VEL
LIN {X 0,Y 163.663,Z 800.899,A -85,B 0,C 180,E1 27523.024,E2 27523.024} C_VEL
LIN {X 0,Y 161.931,Z 804.954,A -85,B 0,C 180,E1 27527.393,E2 27527.393} C_VEL
LIN {X 0,Y 110.616,Z 846.319,A -85,B 0,C 180,E1 27532.097,E2 27532.097} C_VEL
LIN {X 0,Y 77.729,Z 864.405,A -85,B 0,C 180,E1 27538.115,E2 27538.115} C_VEL
LIN {X 0,Y 44.324,Z 875.792,A -85,B 0,C 180,E1 27542.253,E2 27542.253} C_VEL
LIN {X 0,Y 15.065,Z 884.297,A -85,B 0,C 180,E1 27599.727,E2 27599.727} C_VEL
LIN {X 0,Y 14.765,Z 885.358,A -85,B 0,C 180,E1 27660.892,E2 27660.892} C_VEL
LIN {X 0,Y 40.696,Z 883.509,A -85,B 0,C 180,E1 27717.225,E2 27717.225} C_VEL
LIN {X 0,Y 30.601,Z 875.613,A -85,B 0,C 180,E1 27843.662,E2 27843.662} C_VEL
LIN {X 0,Y 87.364,Z 854.248,A -85,B 0,C 180,E1 27868.952,E2 27868.952} C_VEL
LIN {X 0,Y 140.45,Z 820.055,A -85,B 0,C 180,E1 27874.815,E2 27874.815} C_VEL
LIN {X 0,Y 156.057,Z 806.445,A -85,B 0,C 180,E1 27876.48,E2 27876.48} C_VEL
LIN {X 0,Y 157.37,Z 807.768,A -85,B 0,C 180,E1 27884.618,E2 27884.618} C_VEL
LIN {X 0,Y 105.302,Z 847.937,A -85,B 0,C 180,E1 27888.39,E2 27888.39} C_VEL
LIN {X 0,Y 48.887,Z 874.245,A -85,B 0,C 180,E1 27900.089,E2 27900.089} C_VEL
LIN {X 0,Y 44.324,Z 875.792,A -85,B 0,C 180,E1 27902.253,E2 27902.253} C_VEL
LIN {X 0,Y 10.361,Z 882.51,A -85,B 0,C 180,E1 27924.996,E2 27924.996} C_VEL
LIN {X 0,Y 8.812,Z 883.966,A -85,B 0,C 180,E1 28049.349,E2 28049.349} C_VEL
LIN {X 0,Y 20.022,Z 883.697,A -85,B 0,C 180,E1 28079.402,E2 28079.402} C_VEL
LIN {X 0,Y 45.446,Z 871.461,A -85,B 0,C 180,E1 28226.609,E2 28226.609} C_VEL
LIN {X 0,Y 103.996,Z 845.751,A -85,B 0,C 180,E1 28235.793,E2 28235.793} C_VEL
LIN {X 0,Y 150.364,Z 812.131,A -85,B 0,C 180,E1 28238.481,E2 28238.481} C_VEL
LIN {X 0,Y 150.757,Z 812.804,A -85,B 0,C 180,E1 28242.013,E2 28242.013} C_VEL
LIN {X 0,Y 99.069,Z 850.234,A -85,B 0,C 180,E1 28244.406,E2 28244.406} C_VEL
LIN {X 0,Y 38.201,Z 875.919,A -85,B 0,C 180,E1 28253.359,E2 28253.359} C_VEL
LIN {X 0,Y 10.361,Z 882.51,A -85,B 0,C 180,E1 28284.996,E2 28284.996} C_VEL
LIN {X 0,Y 15.247,Z 880.335,A -85,B 0,C 180,E1 28247.411,E2 28247.411} C_VEL
LIN {X 0,Y 40.173,Z 873.65,A -85,B 0,C 180,E1 28236.297,E2 28236.297} C_VEL
LIN {X 0,Y 88.829,Z 854.706,A -85,B 0,C 180,E1 28239.997,E2 28239.997} C_VEL
LIN {X 0,Y 28.027,Z 877.309,A -85,B 0,C 180,E1 28241.355,E2 28241.355} C_VEL
LIN {X 0,Y 8.664,Z 881.136,A -85,B 0,C 180,E1 28231.234,E2 28231.234} C_VEL
LIN {X 0,Y 40.173,Z 873.65,A -85,B 0,C 180,E1 28236.297,E2 28236.297} C_VEL
LIN {X 0,Y 42.715,Z 875.574,A -85,B 0,C 180,E1 28236.51,E2 28236.51} C_VEL
LIN {X 0,Y 42.715,Z 951,A -85,B 0,C 180,E1 28236.51,E2 28236.51} C_VEL
LIN {X 0,Y 42.715,Z 951,A -85,B 0,C 180,E1 28236.51,E2 28236.51}

